KUKA KRL program: EPS_2_25252_SD6A_A_20250911081714.src

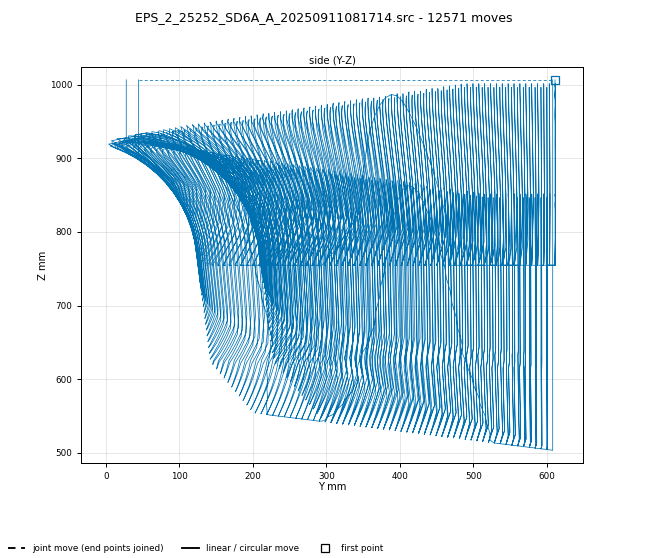
[picture p0: tool path of EPS_2_25252_SD6A_A_20250911081714.src, 12571 of 12573 moves have a stored position in this frame; points joined in program order, loops and branches not executed]
&ACCESS RVP
&REL 4
&COMMENT QRS 19112012
&PARAM EDITMASK = *
DEF PART()
EXT BAS (BAS_COMMAND :IN,REAL :IN )
INT I
BAS (#INITMOV,0 )

;KUKA QRS Post kuka4.cps  Date:22-06-2017 !

File_ID=2841

QRS_PRE_INIT()

;Init var - Until changes are made in qrs_pre_init
Outlet_Square_prg=0
Inlet_1_Square_prg=0
Inlet_2_Square_prg=0
Inlet_3_Square_prg=0
Inlet_4_Square_prg=0
Inlet_5_Square_prg=0

Outlet_1={X 0.000, Y 489.850, Z 814.000, B 0.000, E1 0.000 }
Inlet_1={X 0.000, Y 516.730, Z 721.500, B 0.000, E1 160.000 }
Outlet_1_type=366
Inlet_1_type=201
;QRS#1=Sidecore dimensions
;QRS#2=375-15" PVC SDR 35
;QRS#3=200-8" PVC SDR 35
;QRS#4=
;QRS#5=
;QRS#6=
;QRS#7=
;QRS#8=
;QRS#9=20Y PSX
;QRS#10=12-08 PSX
;QRS#11=
;QRS#12=
;QRS#13=
;QRS#14=
;QRS#15=
;QRS#16=1220x127x1295 4,25'
;QRS#17=EPS Height
;QRS#18=997
;QRS#19=*
;QRS#20= UPDATED VERSION 22-06-2017
;QRS#21=*
Outlet_Square=0250
Inlet_1_Square=0100
Inlet_2_Square=0
Inlet_3_Square=0
Inlet_4_Square=0
Inlet_5_Square=0
Mill_Square=1
Outlet_Square_Prg=252
Inlet_1_Square_prg=204

QRS_INIT()

$ADVANCE=5

; T1
PTP {E1 177.287,E2 177.287}
PTP {X 0,Y 611.066,A -85,B 0,C 180,E1 177.287,E2 177.287,E3 0,E4 0,E5 0,E6 0}
QRS_SPEED_INIT()
LIN {X 0,Y 611.066,Z 1007,A -85,B 0,C 180,E1 177.287,E2 177.287,E3 0,E4 0,E5 0,E6 0} C_VEL
LIN {X 0,Y 611.066,Z 756.81,A -85,B 0,C 180,E1 177.287,E2 177.287} C_VEL
LIN {X 0,Y 611.138,Z 754.81,A -85,B 0,C 180,E1 177.474,E2 177.474} C_VEL
LIN {X 0,Y 611.86,Z 754.81,A -85,B 0,C 180,E1 178.833,E2 178.833} C_VEL
LIN {X 0,Y 611.81,Z 754.81,A -85,B 0,C 180,E1 185.845,E2 185.845} C_VEL
LIN {X 0,Y 611.809,Z 754.81,A -85,B 0,C 180,E1 192.947,E2 192.947} C_VEL
LIN {X 0,Y 611.774,Z 754.81,A -85,B 0,C 180,E1 200.26,E2 200.26} C_VEL
LIN {X 0,Y 611.796,Z 754.81,A -85,B 0,C 180,E1 207.935,E2 207.935} C_VEL
LIN {X 0,Y 610.461,Z 754.81,A -85,B 0,C 180,E1 210.686,E2 210.686} C_VEL
LIN {X 0,Y 611.788,Z 754.81,A -85,B 0,C 180,E1 216.206,E2 216.206} C_VEL
LIN {X 0,Y 611.203,Z 754.81,A -85,B 0,C 180,E1 217.339,E2 217.339} C_VEL
LIN {X 0,Y 610.736,Z 754.81,A -85,B 0,C 180,E1 222.324,E2 222.324} C_VEL
LIN {X 0,Y 611.764,Z 754.81,A -85,B 0,C 180,E1 224.532,E2 224.532} C_VEL
LIN {X 0,Y 611.743,Z 754.81,A -85,B 0,C 180,E1 232.602,E2 232.602} C_VEL
LIN {X 0,Y 611.207,Z 754.81,A -85,B 0,C 180,E1 233.759,E2 233.759} C_VEL
LIN {X 0,Y 611.694,Z 754.81,A -85,B 0,C 180,E1 241.163,E2 241.163} C_VEL
LIN {X 0,Y 611.5,Z 754.81,A -85,B 0,C 180,E1 242.054,E2 242.054} C_VEL
LIN {X 0,Y 611.785,Z 754.81,A -85,B 0,C 180,E1 248.628,E2 248.628} C_VEL
LIN {X 0,Y 610.978,Z 754.81,A -85,B 0,C 180,E1 248.985,E2 248.985} C_VEL
LIN {X 0,Y 610.824,Z 754.81,A -85,B 0,C 180,E1 249.003,E2 249.003} C_VEL
LIN {X 0,Y 611.647,Z 795.005,A -85,B 0,C 180,E1 249.534,E2 249.534} C_VEL
LIN {X 0,Y 611.812,Z 820.275,A -85,B 0,C 180,E1 249.861,E2 249.861} C_VEL
LIN {X 0,Y 611.831,Z 829.389,A -85,B 0,C 180,E1 250.017,E2 250.017} C_VEL
LIN {X 0,Y 611.809,Z 838.409,A -85,B 0,C 180,E1 250.21,E2 250.21} C_VEL
LIN {X 0,Y 611.672,Z 847.342,A -85,B 0,C 180,E1 250.438,E2 250.438} C_VEL
LIN {X 0,Y 611.791,Z 856.186,A -85,B 0,C 180,E1 250.713,E2 250.713} C_VEL
LIN {X 0,Y 611.791,Z 863.938,A -85,B 0,C 180,E1 250.983,E2 250.983} C_VEL
LIN {X 0,Y 611.787,Z 873.56,A -85,B 0,C 180,E1 251.368,E2 251.368} C_VEL
LIN {X 0,Y 611.803,Z 882.055,A -85,B 0,C 180,E1 251.753,E2 251.753} C_VEL
LIN {X 0,Y 611.728,Z 891.103,A -85,B 0,C 180,E1 252.211,E2 252.211} C_VEL
LIN {X 0,Y 611.707,Z 900.538,A -85,B 0,C 180,E1 252.749,E2 252.749} C_VEL
LIN {X 0,Y 611.545,Z 908.953,A -85,B 0,C 180,E1 253.278,E2 253.278} C_VEL
LIN {X 0,Y 611.447,Z 915.387,A -85,B 0,C 180,E1 253.72,E2 253.72} C_VEL
LIN {X 0,Y 611.512,Z 922.82,A -85,B 0,C 180,E1 254.281,E2 254.281} C_VEL
LIN {X 0,Y 611.728,Z 930.719,A -85,B 0,C 180,E1 254.939,E2 254.939} C_VEL
LIN {X 0,Y 611.828,Z 937.206,A -85,B 0,C 180,E1 255.524,E2 255.524} C_VEL
LIN {X 0,Y 611.642,Z 944.107,A -85,B 0,C 180,E1 256.197,E2 256.197} C_VEL
LIN {X 0,Y 611.382,Z 950.111,A -85,B 0,C 180,E1 256.833,E2 256.833} C_VEL
LIN {X 0,Y 611.256,Z 955.826,A -85,B 0,C 180,E1 257.492,E2 257.492} C_VEL
LIN {X 0,Y 611.362,Z 961.718,A -85,B 0,C 180,E1 258.241,E2 258.241} C_VEL
LIN {X 0,Y 611.558,Z 966.083,A -85,B 0,C 180,E1 258.841,E2 258.841} C_VEL
LIN {X 0,Y 611.865,Z 971.956,A -85,B 0,C 180,E1 259.737,E2 259.737} C_VEL
LIN {X 0,Y 611.486,Z 977.196,A -85,B 0,C 180,E1 260.619,E2 260.619} C_VEL
LIN {X 0,Y 611.213,Z 980.408,A -85,B 0,C 180,E1 261.206,E2 261.206} C_VEL
LIN {X 0,Y 611.061,Z 984.692,A -85,B 0,C 180,E1 262.09,E2 262.09} C_VEL
LIN {X 0,Y 611.227,Z 988.443,A -85,B 0,C 180,E1 262.976,E2 262.976} C_VEL
LIN {X 0,Y 611.496,Z 990.636,A -85,B 0,C 180,E1 263.566,E2 263.566} C_VEL
LIN {X 0,Y 611.768,Z 992.621,A -85,B 0,C 180,E1 264.156,E2 264.156} C_VEL
LIN {X 0,Y 611.736,Z 994.457,A -85,B 0,C 180,E1 264.742,E2 264.742} C_VEL
LIN {X 0,Y 611.169,Z 997.433,A -85,B 0,C 180,E1 265.909,E2 265.909} C_VEL
LIN {X 0,Y 610.976,Z 998.684,A -85,B 0,C 180,E1 266.494,E2 266.494} C_VEL
LIN {X 0,Y 611.094,Z 1000.535,A -85,B 0,C 180,E1 267.713,E2 267.713} C_VEL
LIN {X 0,Y 611.599,Z 1001.553,A -85,B 0,C 180,E1 268.834,E2 268.834} C_VEL
LIN {X 0,Y 611.712,Z 1001.903,A -85,B 0,C 180,E1 269.768,E2 269.768} C_VEL
LIN {X 0,Y 611.468,Z 1001.915,A -85,B 0,C 180,E1 270.235,E2 270.235} C_VEL
LIN {X 0,Y 611.076,Z 1001.575,A -85,B 0,C 180,E1 271.17,E2 271.17} C_VEL
LIN {X 0,Y 611.004,Z 1000.586,A -85,B 0,C 180,E1 272.247,E2 272.247} C_VEL
LIN {X 0,Y 611.446,Z 998.665,A -85,B 0,C 180,E1 273.506,E2 273.506} C_VEL
LIN {X 0,Y 611.741,Z 997.407,A -85,B 0,C 180,E1 274.089,E2 274.089} C_VEL
LIN {X 0,Y 611.75,Z 996.021,A -85,B 0,C 180,E1 274.674,E2 274.674} C_VEL
LIN {X 0,Y 611.455,Z 994.46,A -85,B 0,C 180,E1 275.263,E2 275.263} C_VEL
LIN {X 0,Y 611.035,Z 991.688,A -85,B 0,C 180,E1 276.147,E2 276.147} C_VEL
LIN {X 0,Y 610.903,Z 988.434,A -85,B 0,C 180,E1 277.031,E2 277.031} C_VEL
LIN {X 0,Y 611.131,Z 984.681,A -85,B 0,C 180,E1 277.912,E2 277.912} C_VEL
LIN {X 0,Y 611.584,Z 980.396,A -85,B 0,C 180,E1 278.791,E2 278.791} C_VEL
LIN {X 0,Y 611.866,Z 977.182,A -85,B 0,C 180,E1 279.377,E2 279.377} C_VEL
LIN {X 0,Y 611.514,Z 971.941,A -85,B 0,C 180,E1 280.272,E2 280.272} C_VEL
LIN {X 0,Y 611.151,Z 964.994,A -85,B 0,C 180,E1 281.318,E2 281.318} C_VEL
LIN {X 0,Y 611.162,Z 959.425,A -85,B 0,C 180,E1 282.064,E2 282.064} C_VEL
LIN {X 0,Y 611.425,Z 953.292,A -85,B 0,C 180,E1 282.806,E2 282.806} C_VEL
LIN {X 0,Y 611.786,Z 945.803,A -85,B 0,C 180,E1 283.623,E2 283.623} C_VEL
LIN {X 0,Y 611.787,Z 939.857,A -85,B 0,C 180,E1 284.223,E2 284.223} C_VEL
LIN {X 0,Y 611.566,Z 932.74,A -85,B 0,C 180,E1 284.888,E2 284.888} C_VEL
LIN {X 0,Y 611.429,Z 926.124,A -85,B 0,C 180,E1 285.455,E2 285.455} C_VEL
LIN {X 0,Y 611.439,Z 919.137,A -85,B 0,C 180,E1 286.004,E2 286.004} C_VEL
LIN {X 0,Y 611.611,Z 911.498,A -85,B 0,C 180,E1 286.549,E2 286.549} C_VEL
LIN {X 0,Y 611.767,Z 903.322,A -85,B 0,C 180,E1 287.08,E2 287.08} C_VEL
LIN {X 0,Y 611.817,Z 895.304,A -85,B 0,C 180,E1 287.555,E2 287.555} C_VEL
LIN {X 0,Y 611.786,Z 886.651,A -85,B 0,C 180,E1 288.02,E2 288.02} C_VEL
LIN {X 0,Y 611.701,Z 878.735,A -85,B 0,C 180,E1 288.406,E2 288.406} C_VEL
LIN {X 0,Y 611.692,Z 869.834,A -85,B 0,C 180,E1 288.792,E2 288.792} C_VEL
LIN {X 0,Y 611.795,Z 859.549,A -85,B 0,C 180,E1 289.174,E2 289.174} C_VEL
LIN {X 0,Y 611.763,Z 849.942,A -85,B 0,C 180,E1 289.484,E2 289.484} C_VEL
LIN {X 0,Y 611.768,Z 843.149,A -85,B 0,C 180,E1 289.678,E2 289.678} C_VEL
LIN {X 0,Y 611.844,Z 831.276,A -85,B 0,C 180,E1 289.946,E2 289.946} C_VEL
LIN {X 0,Y 611.833,Z 821.432,A -85,B 0,C 180,E1 290.121,E2 290.121} C_VEL
LIN {X 0,Y 611.678,Z 798.302,A -85,B 0,C 180,E1 290.424,E2 290.424} C_VEL
LIN {X 0,Y 610.927,Z 760.221,A -85,B 0,C 180,E1 290.919,E2 290.919} C_VEL
LIN {X 0,Y 610.799,Z 754.81,A -85,B 0,C 180,E1 290.996,E2 290.996} C_VEL
LIN {X 0,Y 611.629,Z 754.81,A -85,B 0,C 180,E1 291.129,E2 291.129} C_VEL
LIN {X 0,Y 611.582,Z 754.81,A -85,B 0,C 180,E1 291.731,E2 291.731} C_VEL
LIN {X 0,Y 611.82,Z 754.81,A -85,B 0,C 180,E1 297.933,E2 297.933} C_VEL
LIN {X 0,Y 610.472,Z 754.81,A -85,B 0,C 180,E1 300.684,E2 300.684} C_VEL
LIN {X 0,Y 611.766,Z 754.81,A -85,B 0,C 180,E1 306.206,E2 306.206} C_VEL
LIN {X 0,Y 611.188,Z 754.81,A -85,B 0,C 180,E1 307.329,E2 307.329} C_VEL
LIN {X 0,Y 610.711,Z 754.81,A -85,B 0,C 180,E1 312.324,E2 312.324} C_VEL
LIN {X 0,Y 611.745,Z 754.81,A -85,B 0,C 180,E1 314.524,E2 314.524} C_VEL
LIN {X 0,Y 611.706,Z 754.81,A -85,B 0,C 180,E1 322.603,E2 322.603} C_VEL
LIN {X 0,Y 611.179,Z 754.81,A -85,B 0,C 180,E1 323.752,E2 323.752} C_VEL
LIN {X 0,Y 611.635,Z 754.81,A -85,B 0,C 180,E1 331.167,E2 331.167} C_VEL
LIN {X 0,Y 611.406,Z 754.81,A -85,B 0,C 180,E1 332.045,E2 332.045} C_VEL
LIN {X 0,Y 611.799,Z 754.81,A -85,B 0,C 180,E1 339.741,E2 339.741} C_VEL
LIN {X 0,Y 611.858,Z 754.81,A -85,B 0,C 180,E1 347.054,E2 347.054} C_VEL
LIN {X 0,Y 611.817,Z 754.81,A -85,B 0,C 180,E1 354.155,E2 354.155} C_VEL
LIN {X 0,Y 611.87,Z 754.81,A -85,B 0,C 180,E1 361.167,E2 361.167} C_VEL
LIN {X 0,Y 611.807,Z 754.81,A -85,B 0,C 180,E1 368.197,E2 368.197} C_VEL
LIN {X 0,Y 611.836,Z 754.81,A -85,B 0,C 180,E1 375.353,E2 375.353} C_VEL
LIN {X 0,Y 611.769,Z 754.81,A -85,B 0,C 180,E1 382.769,E2 382.769} C_VEL
LIN {X 0,Y 611.754,Z 754.81,A -85,B 0,C 180,E1 390.614,E2 390.614} C_VEL
LIN {X 0,Y 611.703,Z 754.81,A -85,B 0,C 180,E1 399.162,E2 399.162} C_VEL
LIN {X 0,Y 610.297,Z 754.81,A -85,B 0,C 180,E1 402.362,E2 402.362} C_VEL
LIN {X 0,Y 610.609,Z 754.81,A -85,B 0,C 180,E1 405.585,E2 405.585} C_VEL
LIN {X 0,Y 611.693,Z 754.81,A -85,B 0,C 180,E1 407.76,E2 407.76} C_VEL
LIN {X 0,Y 610.234,Z 754.81,A -85,B 0,C 180,E1 413.689,E2 413.689} C_VEL
LIN {X 0,Y 611.762,Z 754.81,A -85,B 0,C 180,E1 416.636,E2 416.636} C_VEL
LIN {X 0,Y 611.77,Z 754.81,A -85,B 0,C 180,E1 424.676,E2 424.676} C_VEL
LIN {X 0,Y 611.495,Z 754.81,A -85,B 0,C 180,E1 433.294,E2 433.294} C_VEL
LIN {X 0,Y 611.27,Z 754.81,A -85,B 0,C 180,E1 434.632,E2 434.632} C_VEL
LIN {X 0,Y 611.862,Z 754.81,A -85,B 0,C 180,E1 441.803,E2 441.803} C_VEL
LIN {X 0,Y 611.873,Z 754.81,A -85,B 0,C 180,E1 448.832,E2 448.832} C_VEL
LIN {X 0,Y 611.829,Z 754.81,A -85,B 0,C 180,E1 457.975,E2 457.975} C_VEL
LIN {X 0,Y 611.668,Z 754.904,A -85,B 0,C 180,E1 458.053,E2 458.053} C_VEL
LIN {X 0,Y 611.818,Z 763.461,A -85,B 0,C 180,E1 458.305,E2 458.305} C_VEL
LIN {X 0,Y 611.721,Z 770.819,A -85,B 0,C 180,E1 458.565,E2 458.565} C_VEL
LIN {X 0,Y 611.704,Z 779.374,A -85,B 0,C 180,E1 458.934,E2 458.934} C_VEL
LIN {X 0,Y 611.785,Z 786.58,A -85,B 0,C 180,E1 459.302,E2 459.302} C_VEL
LIN {X 0,Y 611.823,Z 794.066,A -85,B 0,C 180,E1 459.745,E2 459.745} C_VEL
LIN {X 0,Y 611.7,Z 801.675,A -85,B 0,C 180,E1 460.266,E2 460.266} C_VEL
LIN {X 0,Y 611.527,Z 809.163,A -85,B 0,C 180,E1 460.863,E2 460.863} C_VEL
LIN {X 0,Y 611.583,Z 813.985,A -85,B 0,C 180,E1 461.308,E2 461.308} C_VEL
LIN {X 0,Y 611.754,Z 819.881,A -85,B 0,C 180,E1 461.9,E2 461.9} C_VEL
LIN {X 0,Y 611.847,Z 825.006,A -85,B 0,C 180,E1 462.495,E2 462.495} C_VEL
LIN {X 0,Y 611.571,Z 830.05,A -85,B 0,C 180,E1 463.153,E2 463.153} C_VEL
LIN {X 0,Y 611.352,Z 834.118,A -85,B 0,C 180,E1 463.768,E2 463.768} C_VEL
LIN {X 0,Y 611.348,Z 837.585,A -85,B 0,C 180,E1 464.364,E2 464.364} C_VEL
LIN {X 0,Y 611.521,Z 840.61,A -85,B 0,C 180,E1 464.959,E2 464.959} C_VEL
LIN {X 0,Y 611.855,Z 843.98,A -85,B 0,C 180,E1 465.744,E2 465.744} C_VEL
LIN {X 0,Y 611.76,Z 845.466,A -85,B 0,C 180,E1 466.141,E2 466.141} C_VEL
LIN {X 0,Y 611.48,Z 847.279,A -85,B 0,C 180,E1 466.702,E2 466.702} C_VEL
LIN {X 0,Y 611.285,Z 848.511,A -85,B 0,C 180,E1 467.155,E2 467.155} C_VEL
LIN {X 0,Y 611.186,Z 849.953,A -85,B 0,C 180,E1 467.805,E2 467.805} C_VEL
LIN {X 0,Y 611.315,Z 850.927,A -85,B 0,C 180,E1 468.416,E2 468.416} C_VEL
LIN {X 0,Y 611.592,Z 851.56,A -85,B 0,C 180,E1 469.024,E2 469.024} C_VEL
LIN {X 0,Y 611.86,Z 851.874,A -85,B 0,C 180,E1 469.633,E2 469.633} C_VEL
LIN {X 0,Y 611.627,Z 851.891,A -85,B 0,C 180,E1 470.262,E2 470.262} C_VEL
LIN {X 0,Y 611.328,Z 851.62,A -85,B 0,C 180,E1 470.821,E2 470.821} C_VEL
LIN {X 0,Y 611.148,Z 851.071,A -85,B 0,C 180,E1 471.378,E2 471.378} C_VEL
LIN {X 0,Y 611.149,Z 849.995,A -85,B 0,C 180,E1 472.081,E2 472.081} C_VEL
LIN {X 0,Y 611.419,Z 848.438,A -85,B 0,C 180,E1 472.78,E2 472.78} C_VEL
LIN {X 0,Y 611.84,Z 846.085,A -85,B 0,C 180,E1 473.578,E2 473.578} C_VEL
LIN {X 0,Y 611.755,Z 844.446,A -85,B 0,C 180,E1 474.043,E2 474.043} C_VEL
LIN {X 0,Y 611.36,Z 840.812,A -85,B 0,C 180,E1 474.912,E2 474.912} C_VEL
LIN {X 0,Y 611.234,Z 837.514,A -85,B 0,C 180,E1 475.56,E2 475.56} C_VEL
LIN {X 0,Y 611.357,Z 833.768,A -85,B 0,C 180,E1 476.199,E2 476.199} C_VEL
LIN {X 0,Y 611.664,Z 829.491,A -85,B 0,C 180,E1 476.833,E2 476.833} C_VEL
LIN {X 0,Y 611.854,Z 826.255,A -85,B 0,C 180,E1 477.262,E2 477.262} C_VEL
LIN {X 0,Y 611.7,Z 820.546,A -85,B 0,C 180,E1 477.936,E2 477.936} C_VEL
LIN {X 0,Y 611.506,Z 814.309,A -85,B 0,C 180,E1 478.572,E2 478.572} C_VEL
LIN {X 0,Y 611.468,Z 809.884,A -85,B 0,C 180,E1 478.986,E2 478.986} C_VEL
LIN {X 0,Y 611.642,Z 803.331,A -85,B 0,C 180,E1 479.52,E2 479.52} C_VEL
LIN {X 0,Y 611.818,Z 795.711,A -85,B 0,C 180,E1 480.057,E2 480.057} C_VEL
LIN {X 0,Y 611.78,Z 788.564,A -85,B 0,C 180,E1 480.498,E2 480.498} C_VEL
LIN {X 0,Y 611.615,Z 780.628,A -85,B 0,C 180,E1 480.917,E2 480.917} C_VEL
LIN {X 0,Y 611.602,Z 773.495,A -85,B 0,C 180,E1 481.239,E2 481.239} C_VEL
LIN {X 0,Y 611.747,Z 764.95,A -85,B 0,C 180,E1 481.558,E2 481.558} C_VEL
LIN {X 0,Y 611.758,Z 755.735,A -85,B 0,C 180,E1 481.833,E2 481.833} C_VEL
LIN {X 0,Y 611.697,Z 754.81,A -85,B 0,C 180,E1 481.867,E2 481.867} C_VEL
LIN {X 0,Y 611.77,Z 754.81,A -85,B 0,C 180,E1 489.152,E2 489.152} C_VEL
LIN {X 0,Y 610.356,Z 754.81,A -85,B 0,C 180,E1 492.351,E2 492.351} C_VEL
LIN {X 0,Y 610.67,Z 754.81,A -85,B 0,C 180,E1 495.572,E2 495.572} C_VEL
LIN {X 0,Y 611.767,Z 754.81,A -85,B 0,C 180,E1 497.764,E2 497.764} C_VEL
LIN {X 0,Y 610.275,Z 754.81,A -85,B 0,C 180,E1 503.69,E2 503.69} C_VEL
LIN {X 0,Y 611.79,Z 754.81,A -85,B 0,C 180,E1 506.636,E2 506.636} C_VEL
LIN {X 0,Y 611.824,Z 754.81,A -85,B 0,C 180,E1 514.677,E2 514.677} C_VEL
LIN {X 0,Y 611.477,Z 754.81,A -85,B 0,C 180,E1 523.279,E2 523.279} C_VEL
LIN {X 0,Y 611.227,Z 754.81,A -85,B 0,C 180,E1 524.631,E2 524.631} C_VEL
LIN {X 0,Y 611.802,Z 754.81,A -85,B 0,C 180,E1 531.803,E2 531.803} C_VEL
LIN {X 0,Y 611.138,Z 754.81,A -85,B 0,C 180,E1 537.474,E2 537.474} C_VEL
LIN {X 0,Y 602.939,Z 754.81,A -85,B 0,C 180,E1 540.753,E2 540.753} C_VEL
LIN {X 0,Y 602.827,Z 754.81,A -85,B 0,C 180,E1 547.957,E2 547.957} C_VEL
LIN {X 0,Y 602.702,Z 754.81,A -85,B 0,C 180,E1 555.328,E2 555.328} C_VEL
LIN {X 0,Y 603.089,Z 754.81,A -85,B 0,C 180,E1 561.397,E2 561.397} C_VEL
LIN {X 0,Y 602.77,Z 754.81,A -85,B 0,C 180,E1 569.705,E2 569.705} C_VEL
LIN {X 0,Y 603.072,Z 754.81,A -85,B 0,C 180,E1 577.565,E2 577.565} C_VEL
LIN {X 0,Y 602.786,Z 754.81,A -85,B 0,C 180,E1 586.185,E2 586.185} C_VEL
LIN {X 0,Y 603.196,Z 754.81,A -85,B 0,C 180,E1 593.756,E2 593.756} C_VEL
LIN {X 0,Y 602.95,Z 754.81,A -85,B 0,C 180,E1 603.311,E2 603.311} C_VEL
LIN {X 0,Y 603.355,Z 756.25,A -85,B 0,C 180,E1 608.756,E2 608.756} C_VEL
LIN {X 0,Y 604.125,Z 848.863,A -85,B 0,C 180,E1 610.228,E2 610.228} C_VEL
LIN {X 0,Y 603.994,Z 900.949,A -85,B 0,C 180,E1 612.547,E2 612.547} C_VEL
LIN {X 0,Y 603.809,Z 944.075,A -85,B 0,C 180,E1 616.011,E2 616.011} C_VEL
LIN {X 0,Y 603.502,Z 977.731,A -85,B 0,C 180,E1 620.593,E2 620.593} C_VEL
LIN {X 0,Y 603.275,Z 997.05,A -85,B 0,C 180,E1 625.672,E2 625.672} C_VEL
LIN {X 0,Y 603.271,Z 1001.839,A -85,B 0,C 180,E1 630.721,E2 630.721} C_VEL
LIN {X 0,Y 603.203,Z 993.115,A -85,B 0,C 180,E1 635.776,E2 635.776} C_VEL
LIN {X 0,Y 603.407,Z 970.196,A -85,B 0,C 180,E1 640.69,E2 640.69} C_VEL
LIN {X 0,Y 603.74,Z 934.098,A -85,B 0,C 180,E1 644.965,E2 644.965} C_VEL
LIN {X 0,Y 604.102,Z 887.651,A -85,B 0,C 180,E1 648.207,E2 648.207} C_VEL
LIN {X 0,Y 604.321,Z 835.988,A -85,B 0,C 180,E1 650.104,E2 650.104} C_VEL
LIN {X 0,Y 603.622,Z 754.81,A -85,B 0,C 180,E1 651.38,E2 651.38} C_VEL
LIN {X 0,Y 602.793,Z 754.81,A -85,B 0,C 180,E1 659.713,E2 659.713} C_VEL
LIN {X 0,Y 603.053,Z 754.81,A -85,B 0,C 180,E1 667.566,E2 667.566} C_VEL
LIN {X 0,Y 602.757,Z 754.81,A -85,B 0,C 180,E1 676.185,E2 676.185} C_VEL
LIN {X 0,Y 603.175,Z 754.81,A -85,B 0,C 180,E1 683.757,E2 683.757} C_VEL
LIN {X 0,Y 603.254,Z 754.81,A -85,B 0,C 180,E1 692.267,E2 692.267} C_VEL
LIN {X 0,Y 602.853,Z 754.81,A -85,B 0,C 180,E1 701.662,E2 701.662} C_VEL
LIN {X 0,Y 602.898,Z 754.81,A -85,B 0,C 180,E1 709.12,E2 709.12} C_VEL
LIN {X 0,Y 602.842,Z 754.81,A -85,B 0,C 180,E1 716.394,E2 716.394} C_VEL
LIN {X 0,Y 602.808,Z 754.81,A -85,B 0,C 180,E1 723.61,E2 723.61} C_VEL
LIN {X 0,Y 603.164,Z 754.81,A -85,B 0,C 180,E1 729.414,E2 729.414} C_VEL
LIN {X 0,Y 603.021,Z 754.81,A -85,B 0,C 180,E1 736.824,E2 736.824} C_VEL
LIN {X 0,Y 602.77,Z 754.81,A -85,B 0,C 180,E1 744.547,E2 744.547} C_VEL
LIN {X 0,Y 602.582,Z 754.81,A -85,B 0,C 180,E1 752.468,E2 752.468} C_VEL
LIN {X 0,Y 603.22,Z 754.81,A -85,B 0,C 180,E1 759.907,E2 759.907} C_VEL
LIN {X 0,Y 603.356,Z 754.81,A -85,B 0,C 180,E1 768.199,E2 768.199} C_VEL
LIN {X 0,Y 603.218,Z 754.81,A -85,B 0,C 180,E1 777.438,E2 777.438} C_VEL
LIN {X 0,Y 603.153,Z 754.81,A -85,B 0,C 180,E1 785.471,E2 785.471} C_VEL
LIN {X 0,Y 603.238,Z 754.81,A -85,B 0,C 180,E1 794.683,E2 794.683} C_VEL
LIN {X 0,Y 602.911,Z 754.81,A -85,B 0,C 180,E1 803.858,E2 803.858} C_VEL
LIN {X 0,Y 602.597,Z 754.81,A -85,B 0,C 180,E1 810.721,E2 810.721} C_VEL
LIN {X 0,Y 603.88,Z 756.612,A -85,B 0,C 180,E1 817.944,E2 817.944} C_VEL
LIN {X 0,Y 603.91,Z 796.409,A -85,B 0,C 180,E1 819.765,E2 819.765} C_VEL
LIN {X 0,Y 603.782,Z 827.416,A -85,B 0,C 180,E1 822.704,E2 822.704} C_VEL
LIN {X 0,Y 603.602,Z 846.583,A -85,B 0,C 180,E1 826.43,E2 826.43} C_VEL
LIN {X 0,Y 603.782,Z 851.979,A -85,B 0,C 180,E1 829.835,E2 829.835} C_VEL
LIN {X 0,Y 603.782,Z 845.084,A -85,B 0,C 180,E1 833.93,E2 833.93} C_VEL
LIN {X 0,Y 603.788,Z 823.442,A -85,B 0,C 180,E1 837.709,E2 837.709} C_VEL
LIN {X 0,Y 603.91,Z 790.475,A -85,B 0,C 180,E1 840.522,E2 840.522} C_VEL
LIN {X 0,Y 603.494,Z 754.81,A -85,B 0,C 180,E1 842.194,E2 842.194} C_VEL
LIN {X 0,Y 603.287,Z 754.81,A -85,B 0,C 180,E1 849.9,E2 849.9} C_VEL
LIN {X 0,Y 603.418,Z 754.81,A -85,B 0,C 180,E1 858.204,E2 858.204} C_VEL
LIN {X 0,Y 603.274,Z 754.81,A -85,B 0,C 180,E1 867.427,E2 867.427} C_VEL
LIN {X 0,Y 603.227,Z 754.81,A -85,B 0,C 180,E1 875.473,E2 875.473} C_VEL
LIN {X 0,Y 603.194,Z 754.81,A -85,B 0,C 180,E1 884.681,E2 884.681} C_VEL
LIN {X 0,Y 602.878,Z 754.81,A -85,B 0,C 180,E1 893.875,E2 893.875} C_VEL
LIN {X 0,Y 602.939,Z 754.81,A -85,B 0,C 180,E1 900.753,E2 900.753} C_VEL
LIN {X 0,Y 594.952,Z 754.81,A -85,B 0,C 180,E1 904.052,E2 904.052} C_VEL
LIN {X 0,Y 595.421,Z 754.81,A -85,B 0,C 180,E1 912.51,E2 912.51} C_VEL
LIN {X 0,Y 594.956,Z 754.81,A -85,B 0,C 180,E1 921.704,E2 921.704} C_VEL
LIN {X 0,Y 594.736,Z 754.81,A -85,B 0,C 180,E1 929.837,E2 929.837} C_VEL
LIN {X 0,Y 595.425,Z 754.81,A -85,B 0,C 180,E1 936.792,E2 936.792} C_VEL
LIN {X 0,Y 595.044,Z 754.81,A -85,B 0,C 180,E1 945.465,E2 945.465} C_VEL
LIN {X 0,Y 595.255,Z 754.81,A -85,B 0,C 180,E1 953.421,E2 953.421} C_VEL
LIN {X 0,Y 595.313,Z 754.81,A -85,B 0,C 180,E1 961.862,E2 961.862} C_VEL
LIN {X 0,Y 595.708,Z 756.326,A -85,B 0,C 180,E1 968.471,E2 968.471} C_VEL
LIN {X 0,Y 596.585,Z 848.864,A -85,B 0,C 180,E1 969.967,E2 969.967} C_VEL
LIN {X 0,Y 596.304,Z 900.979,A -85,B 0,C 180,E1 972.316,E2 972.316} C_VEL
LIN {X 0,Y 595.976,Z 944.04,A -85,B 0,C 180,E1 975.82,E2 975.82} C_VEL
LIN {X 0,Y 595.729,Z 975.748,A -85,B 0,C 180,E1 980.099,E2 980.099} C_VEL
LIN {X 0,Y 595.635,Z 995.224,A -85,B 0,C 180,E1 984.884,E2 984.884} C_VEL
LIN {X 0,Y 595.643,Z 1001.839,A -85,B 0,C 180,E1 989.271,E2 989.271} C_VEL
LIN {X 0,Y 595.742,Z 997.049,A -85,B 0,C 180,E1 994.383,E2 994.383} C_VEL
LIN {X 0,Y 595.9,Z 977.727,A -85,B 0,C 180,E1 999.529,E2 999.529} C_VEL
LIN {X 0,Y 596.013,Z 945.729,A -85,B 0,C 180,E1 1003.999,E2 1003.999} C_VEL
LIN {X 0,Y 596.367,Z 901.589,A -85,B 0,C 180,E1 1007.644,E2 1007.644} C_VEL
LIN {X 0,Y 596.659,Z 850.037,A -85,B 0,C 180,E1 1009.995,E2 1009.995} C_VEL
LIN {X 0,Y 595.986,Z 759.919,A -85,B 0,C 180,E1 1011.473,E2 1011.473} C_VEL
LIN {X 0,Y 595.487,Z 754.81,A -85,B 0,C 180,E1 1011.687,E2 1011.687} C_VEL
LIN {X 0,Y 594.758,Z 754.81,A -85,B 0,C 180,E1 1019.839,E2 1019.839} C_VEL
LIN {X 0,Y 595.42,Z 754.81,A -85,B 0,C 180,E1 1026.796,E2 1026.796} C_VEL
LIN {X 0,Y 595.018,Z 754.81,A -85,B 0,C 180,E1 1035.466,E2 1035.466} C_VEL
LIN {X 0,Y 595.232,Z 754.81,A -85,B 0,C 180,E1 1043.429,E2 1043.429} C_VEL
LIN {X 0,Y 595.205,Z 754.81,A -85,B 0,C 180,E1 1051.859,E2 1051.859} C_VEL
LIN {X 0,Y 594.941,Z 754.81,A -85,B 0,C 180,E1 1061.409,E2 1061.409} C_VEL
LIN {X 0,Y 594.918,Z 754.81,A -85,B 0,C 180,E1 1069.144,E2 1069.144} C_VEL
LIN {X 0,Y 594.853,Z 754.81,A -85,B 0,C 180,E1 1076.345,E2 1076.345} C_VEL
LIN {X 0,Y 594.797,Z 754.81,A -85,B 0,C 180,E1 1083.659,E2 1083.659} C_VEL
LIN {X 0,Y 594.754,Z 754.81,A -85,B 0,C 180,E1 1090.773,E2 1090.773} C_VEL
LIN {X 0,Y 594.921,Z 754.81,A -85,B 0,C 180,E1 1097.06,E2 1097.06} C_VEL
LIN {X 0,Y 594.608,Z 754.81,A -85,B 0,C 180,E1 1105.035,E2 1105.035} C_VEL
LIN {X 0,Y 595.098,Z 754.81,A -85,B 0,C 180,E1 1111.52,E2 1111.52} C_VEL
LIN {X 0,Y 594.624,Z 754.81,A -85,B 0,C 180,E1 1121.158,E2 1121.158} C_VEL
LIN {X 0,Y 594.642,Z 754.81,A -85,B 0,C 180,E1 1129.399,E2 1129.399} C_VEL
LIN {X 0,Y 594.722,Z 754.81,A -85,B 0,C 180,E1 1138.459,E2 1138.459} C_VEL
LIN {X 0,Y 594.469,Z 754.81,A -85,B 0,C 180,E1 1146.691,E2 1146.691} C_VEL
LIN {X 0,Y 595.236,Z 754.81,A -85,B 0,C 180,E1 1154.472,E2 1154.472} C_VEL
LIN {X 0,Y 595.047,Z 754.81,A -85,B 0,C 180,E1 1163.409,E2 1163.409} C_VEL
LIN {X 0,Y 594.586,Z 754.81,A -85,B 0,C 180,E1 1170.731,E2 1170.731} C_VEL
LIN {X 0,Y 595.813,Z 756.512,A -85,B 0,C 180,E1 1177.776,E2 1177.776} C_VEL
LIN {X 0,Y 596.015,Z 796.255,A -85,B 0,C 180,E1 1179.618,E2 1179.618} C_VEL
LIN {X 0,Y 595.814,Z 828.021,A -85,B 0,C 180,E1 1182.69,E2 1182.69} C_VEL
LIN {X 0,Y 595.5,Z 847.425,A -85,B 0,C 180,E1 1186.66,E2 1186.66} C_VEL
LIN {X 0,Y 595.63,Z 851.97,A -85,B 0,C 180,E1 1190.118,E2 1190.118} C_VEL
LIN {X 0,Y 595.655,Z 843.869,A -85,B 0,C 180,E1 1194.318,E2 1194.318} C_VEL
LIN {X 0,Y 595.748,Z 820.861,A -85,B 0,C 180,E1 1198.115,E2 1198.115} C_VEL
LIN {X 0,Y 595.954,Z 786.961,A -85,B 0,C 180,E1 1200.873,E2 1200.873} C_VEL
LIN {X 0,Y 595.408,Z 754.81,A -85,B 0,C 180,E1 1202.342,E2 1202.342} C_VEL
LIN {X 0,Y 594.679,Z 754.81,A -85,B 0,C 180,E1 1211.163,E2 1211.163} C_VEL
LIN {X 0,Y 594.689,Z 754.81,A -85,B 0,C 180,E1 1219.402,E2 1219.402} C_VEL
LIN {X 0,Y 594.782,Z 754.81,A -85,B 0,C 180,E1 1228.461,E2 1228.461} C_VEL
LIN {X 0,Y 594.507,Z 754.81,A -85,B 0,C 180,E1 1236.691,E2 1236.691} C_VEL
LIN {X 0,Y 595.199,Z 754.81,A -85,B 0,C 180,E1 1244.47,E2 1244.47} C_VEL
LIN {X 0,Y 595.012,Z 754.81,A -85,B 0,C 180,E1 1253.408,E2 1253.408} C_VEL
LIN {X 0,Y 594.958,Z 754.81,A -85,B 0,C 180,E1 1260.731,E2 1260.731} C_VEL
LIN {X 0,Y 594.952,Z 754.81,A -85,B 0,C 180,E1 1264.052,E2 1264.052} C_VEL
LIN {X 0,Y 587.035,Z 754.81,A -85,B 0,C 180,E1 1267.425,E2 1267.425} C_VEL
LIN {X 0,Y 587.105,Z 754.81,A -85,B 0,C 180,E1 1274.232,E2 1274.232} C_VEL
LIN {X 0,Y 586.825,Z 754.81,A -85,B 0,C 180,E1 1282.021,E2 1282.021} C_VEL
LIN {X 0,Y 586.579,Z 754.81,A -85,B 0,C 180,E1 1290.295,E2 1290.295} C_VEL
LIN {X 0,Y 586.872,Z 754.81,A -85,B 0,C 180,E1 1297.937,E2 1297.937} C_VEL
LIN {X 0,Y 586.578,Z 754.81,A -85,B 0,C 180,E1 1306.718,E2 1306.718} C_VEL
LIN {X 0,Y 586.764,Z 754.81,A -85,B 0,C 180,E1 1314.553,E2 1314.553} C_VEL
LIN {X 0,Y 586.949,Z 754.81,A -85,B 0,C 180,E1 1323.12,E2 1323.12} C_VEL
LIN {X 0,Y 587.567,Z 756.444,A -85,B 0,C 180,E1 1328.159,E2 1328.159} C_VEL
LIN {X 0,Y 589.058,Z 849.901,A -85,B 0,C 180,E1 1329.731,E2 1329.731} C_VEL
LIN {X 0,Y 588.579,Z 901.19,A -85,B 0,C 180,E1 1332.089,E2 1332.089} C_VEL
LIN {X 0,Y 588.134,Z 944.29,A -85,B 0,C 180,E1 1335.654,E2 1335.654} C_VEL
LIN {X 0,Y 587.65,Z 977.732,A -85,B 0,C 180,E1 1340.337,E2 1340.337} C_VEL
LIN {X 0,Y 587.32,Z 997.051,A -85,B 0,C 180,E1 1345.555,E2 1345.555} C_VEL
LIN {X 0,Y 587.26,Z 1001.839,A -85,B 0,C 180,E1 1350.741,E2 1350.741} C_VEL
LIN {X 0,Y 587.241,Z 993.533,A -85,B 0,C 180,E1 1355.798,E2 1355.798} C_VEL
LIN {X 0,Y 587.505,Z 971.486,A -85,B 0,C 180,E1 1360.775,E2 1360.775} C_VEL
LIN {X 0,Y 588.046,Z 935.848,A -85,B 0,C 180,E1 1365.21,E2 1365.21} C_VEL
LIN {X 0,Y 588.767,Z 889.465,A -85,B 0,C 180,E1 1368.601,E2 1368.601} C_VEL
LIN {X 0,Y 589.291,Z 837.458,A -85,B 0,C 180,E1 1370.603,E2 1370.603} C_VEL
LIN {X 0,Y 587.351,Z 754.81,A -85,B 0,C 180,E1 1372.003,E2 1372.003} C_VEL
LIN {X 0,Y 586.622,Z 754.81,A -85,B 0,C 180,E1 1380.296,E2 1380.296} C_VEL
LIN {X 0,Y 586.86,Z 754.81,A -85,B 0,C 180,E1 1387.94,E2 1387.94} C_VEL
LIN {X 0,Y 586.55,Z 754.81,A -85,B 0,C 180,E1 1396.718,E2 1396.718} C_VEL
LIN {X 0,Y 586.717,Z 754.81,A -85,B 0,C 180,E1 1404.565,E2 1404.565} C_VEL
LIN {X 0,Y 586.719,Z 754.81,A -85,B 0,C 180,E1 1413.172,E2 1413.172} C_VEL
LIN {X 0,Y 586.99,Z 754.81,A -85,B 0,C 180,E1 1421.148,E2 1421.148} C_VEL
LIN {X 0,Y 586.996,Z 754.81,A -85,B 0,C 180,E1 1428.822,E2 1428.822} C_VEL
LIN {X 0,Y 586.863,Z 754.81,A -85,B 0,C 180,E1 1436.295,E2 1436.295} C_VEL
LIN {X 0,Y 586.788,Z 754.81,A -85,B 0,C 180,E1 1443.709,E2 1443.709} C_VEL
LIN {X 0,Y 587.08,Z 754.81,A -85,B 0,C 180,E1 1449.675,E2 1449.675} C_VEL
LIN {X 0,Y 586.837,Z 754.81,A -85,B 0,C 180,E1 1457.303,E2 1457.303} C_VEL
LIN {X 0,Y 586.552,Z 754.81,A -85,B 0,C 180,E1 1465.273,E2 1465.273} C_VEL
LIN {X 0,Y 586.481,Z 754.81,A -85,B 0,C 180,E1 1472.757,E2 1472.757} C_VEL
LIN {X 0,Y 586.582,Z 754.81,A -85,B 0,C 180,E1 1481.28,E2 1481.28} C_VEL
LIN {X 0,Y 586.979,Z 754.81,A -85,B 0,C 180,E1 1488.755,E2 1488.755} C_VEL
LIN {X 0,Y 586.793,Z 754.81,A -85,B 0,C 180,E1 1497.982,E2 1497.982} C_VEL
LIN {X 0,Y 586.445,Z 754.81,A -85,B 0,C 180,E1 1506.732,E2 1506.732} C_VEL
LIN {X 0,Y 587.211,Z 754.81,A -85,B 0,C 180,E1 1514.254,E2 1514.254} C_VEL
LIN {X 0,Y 587.076,Z 754.81,A -85,B 0,C 180,E1 1523.32,E2 1523.32} C_VEL
LIN {X 0,Y 586.573,Z 754.81,A -85,B 0,C 180,E1 1530.741,E2 1530.741} C_VEL
LIN {X 0,Y 587.516,Z 755.536,A -85,B 0,C 180,E1 1537.573,E2 1537.573} C_VEL
LIN {X 0,Y 588.143,Z 796.092,A -85,B 0,C 180,E1 1539.467,E2 1539.467} C_VEL
LIN {X 0,Y 587.93,Z 827.248,A -85,B 0,C 180,E1 1542.484,E2 1542.484} C_VEL
LIN {X 0,Y 587.586,Z 847.03,A -85,B 0,C 180,E1 1546.478,E2 1546.478} C_VEL
LIN {X 0,Y 587.515,Z 851.904,A -85,B 0,C 180,E1 1550.408,E2 1550.408} C_VEL
LIN {X 0,Y 587.62,Z 843.766,A -85,B 0,C 180,E1 1554.406,E2 1554.406} C_VEL
LIN {X 0,Y 587.791,Z 821.637,A -85,B 0,C 180,E1 1558.137,E2 1558.137} C_VEL
LIN {X 0,Y 588.062,Z 787.082,A -85,B 0,C 180,E1 1561.015,E2 1561.015} C_VEL
LIN {X 0,Y 587.36,Z 754.81,A -85,B 0,C 180,E1 1562.41,E2 1562.41} C_VEL
LIN {X 0,Y 586.64,Z 754.81,A -85,B 0,C 180,E1 1571.273,E2 1571.273} C_VEL
LIN {X 0,Y 587.064,Z 754.81,A -85,B 0,C 180,E1 1578.761,E2 1578.761} C_VEL
LIN {X 0,Y 586.843,Z 754.81,A -85,B 0,C 180,E1 1587.984,E2 1587.984} C_VEL
LIN {X 0,Y 586.489,Z 754.81,A -85,B 0,C 180,E1 1596.719,E2 1596.719} C_VEL
LIN {X 0,Y 587.177,Z 754.81,A -85,B 0,C 180,E1 1604.252,E2 1604.252} C_VEL
LIN {X 0,Y 587.045,Z 754.81,A -85,B 0,C 180,E1 1613.318,E2 1613.318} C_VEL
LIN {X 0,Y 586.953,Z 754.81,A -85,B 0,C 180,E1 1620.739,E2 1620.739} C_VEL
LIN {X 0,Y 587.035,Z 754.81,A -85,B 0,C 180,E1 1627.425,E2 1627.425} C_VEL
LIN {X 0,Y 578.821,Z 754.81,A -85,B 0,C 180,E1 1630.811,E2 1630.811} C_VEL
LIN {X 0,Y 579.054,Z 754.81,A -85,B 0,C 180,E1 1639.121,E2 1639.121} C_VEL
LIN {X 0,Y 579.026,Z 754.81,A -85,B 0,C 180,E1 1649.001,E2 1649.001} C_VEL
LIN {X 0,Y 578.852,Z 754.81,A -85,B 0,C 180,E1 1658.029,E2 1658.029} C_VEL
LIN {X 0,Y 578.746,Z 754.81,A -85,B 0,C 180,E1 1666.141,E2 1666.141} C_VEL
LIN {X 0,Y 578.844,Z 754.81,A -85,B 0,C 180,E1 1673.851,E2 1673.851} C_VEL
LIN {X 0,Y 578.988,Z 754.81,A -85,B 0,C 180,E1 1682.698,E2 1682.698} C_VEL
LIN {X 0,Y 579.35,Z 755.953,A -85,B 0,C 180,E1 1687.826,E2 1687.826} C_VEL
LIN {X 0,Y 581.581,Z 848.986,A -85,B 0,C 180,E1 1689.431,E2 1689.431} C_VEL
LIN {X 0,Y 580.89,Z 900.956,A -85,B 0,C 180,E1 1691.829,E2 1691.829} C_VEL
LIN {X 0,Y 580.283,Z 944.638,A -85,B 0,C 180,E1 1695.494,E2 1695.494} C_VEL
LIN {X 0,Y 579.711,Z 977.733,A -85,B 0,C 180,E1 1700.203,E2 1700.203} C_VEL
LIN {X 0,Y 579.367,Z 997.05,A -85,B 0,C 180,E1 1705.493,E2 1705.493} C_VEL
LIN {X 0,Y 579.265,Z 1001.838,A -85,B 0,C 180,E1 1710.751,E2 1710.751} C_VEL
LIN {X 0,Y 579.204,Z 993.534,A -85,B 0,C 180,E1 1715.879,E2 1715.879} C_VEL
LIN {X 0,Y 579.477,Z 970.786,A -85,B 0,C 180,E1 1721.043,E2 1721.043} C_VEL
LIN {X 0,Y 580.199,Z 934.751,A -85,B 0,C 180,E1 1725.527,E2 1725.527} C_VEL
LIN {X 0,Y 581.132,Z 887.661,A -85,B 0,C 180,E1 1728.954,E2 1728.954} C_VEL
LIN {X 0,Y 581.823,Z 834.061,A -85,B 0,C 180,E1 1730.965,E2 1730.965} C_VEL
LIN {X 0,Y 579.281,Z 754.81,A -85,B 0,C 180,E1 1732.231,E2 1732.231} C_VEL
LIN {X 0,Y 578.477,Z 754.81,A -85,B 0,C 180,E1 1740.769,E2 1740.769} C_VEL
LIN {X 0,Y 578.838,Z 754.81,A -85,B 0,C 180,E1 1748.033,E2 1748.033} C_VEL
LIN {X 0,Y 578.727,Z 754.81,A -85,B 0,C 180,E1 1756.148,E2 1756.148} C_VEL
LIN {X 0,Y 578.807,Z 754.81,A -85,B 0,C 180,E1 1763.851,E2 1763.851} C_VEL
LIN {X 0,Y 578.793,Z 754.81,A -85,B 0,C 180,E1 1772.69,E2 1772.69} C_VEL
LIN {X 0,Y 579.08,Z 754.81,A -85,B 0,C 180,E1 1780.88,E2 1780.88} C_VEL
LIN {X 0,Y 578.81,Z 754.81,A -85,B 0,C 180,E1 1789.488,E2 1789.488} C_VEL
LIN {X 0,Y 578.9,Z 754.81,A -85,B 0,C 180,E1 1796.244,E2 1796.244} C_VEL
LIN {X 0,Y 578.809,Z 754.81,A -85,B 0,C 180,E1 1803.76,E2 1803.76} C_VEL
LIN {X 0,Y 578.683,Z 754.81,A -85,B 0,C 180,E1 1811.345,E2 1811.345} C_VEL
LIN {X 0,Y 578.789,Z 754.81,A -85,B 0,C 180,E1 1817.551,E2 1817.551} C_VEL
LIN {X 0,Y 578.478,Z 754.81,A -85,B 0,C 180,E1 1825.651,E2 1825.651} C_VEL
LIN {X 0,Y 578.574,Z 754.81,A -85,B 0,C 180,E1 1832.529,E2 1832.529} C_VEL
LIN {X 0,Y 578.49,Z 754.81,A -85,B 0,C 180,E1 1841.612,E2 1841.612} C_VEL
LIN {X 0,Y 578.393,Z 754.81,A -85,B 0,C 180,E1 1849.997,E2 1849.997} C_VEL
LIN {X 0,Y 578.617,Z 754.81,A -85,B 0,C 180,E1 1858.475,E2 1858.475} C_VEL
LIN {X 0,Y 578.673,Z 754.81,A -85,B 0,C 180,E1 1866.015,E2 1866.015} C_VEL
LIN {X 0,Y 578.765,Z 754.81,A -85,B 0,C 180,E1 1875.575,E2 1875.575} C_VEL
LIN {X 0,Y 579.096,Z 754.81,A -85,B 0,C 180,E1 1883.227,E2 1883.227} C_VEL
LIN {X 0,Y 578.56,Z 754.81,A -85,B 0,C 180,E1 1890.751,E2 1890.751} C_VEL
LIN {X 0,Y 579.544,Z 756.488,A -85,B 0,C 180,E1 1897.428,E2 1897.428} C_VEL
LIN {X 0,Y 580.227,Z 797.325,A -85,B 0,C 180,E1 1899.408,E2 1899.408} C_VEL
LIN {X 0,Y 579.833,Z 829.239,A -85,B 0,C 180,E1 1902.661,E2 1902.661} C_VEL
LIN {X 0,Y 579.579,Z 847.25,A -85,B 0,C 180,E1 1906.504,E2 1906.504} C_VEL
LIN {X 0,Y 579.427,Z 851.758,A -85,B 0,C 180,E1 1910.706,E2 1910.706} C_VEL
LIN {X 0,Y 579.405,Z 841.642,A -85,B 0,C 180,E1 1914.998,E2 1914.998} C_VEL
LIN {X 0,Y 579.774,Z 817.414,A -85,B 0,C 180,E1 1918.731,E2 1918.731} C_VEL
LIN {X 0,Y 580.152,Z 782.28,A -85,B 0,C 180,E1 1921.436,E2 1921.436} C_VEL
LIN {X 0,Y 579.231,Z 754.81,A -85,B 0,C 180,E1 1922.69,E2 1922.69} C_VEL
LIN {X 0,Y 578.54,Z 754.81,A -85,B 0,C 180,E1 1931.616,E2 1931.616} C_VEL
LIN {X 0,Y 578.434,Z 754.81,A -85,B 0,C 180,E1 1939.999,E2 1939.999} C_VEL
LIN {X 0,Y 578.669,Z 754.81,A -85,B 0,C 180,E1 1948.464,E2 1948.464} C_VEL
LIN {X 0,Y 578.715,Z 754.81,A -85,B 0,C 180,E1 1956.016,E2 1956.016} C_VEL
LIN {X 0,Y 578.734,Z 754.81,A -85,B 0,C 180,E1 1965.573,E2 1965.573} C_VEL
LIN {X 0,Y 579.064,Z 754.81,A -85,B 0,C 180,E1 1973.225,E2 1973.225} C_VEL
LIN {X 0,Y 578.974,Z 754.81,A -85,B 0,C 180,E1 1980.749,E2 1980.749} C_VEL
LIN {X 0,Y 578.766,Z 754.81,A -85,B 0,C 180,E1 1988.29,E2 1988.29} C_VEL
LIN {X 0,Y 578.821,Z 754.81,A -85,B 0,C 180,E1 1990.811,E2 1990.811} C_VEL
LIN {X 0,Y 571.03,Z 754.81,A -85,B 0,C 180,E1 1994.284,E2 1994.284} C_VEL
LIN {X 0,Y 570.642,Z 754.81,A -85,B 0,C 180,E1 2002.679,E2 2002.679} C_VEL
LIN {X 0,Y 570.599,Z 754.81,A -85,B 0,C 180,E1 2010.189,E2 2010.189} C_VEL
LIN {X 0,Y 570.64,Z 754.81,A -85,B 0,C 180,E1 2018.676,E2 2018.676} C_VEL
LIN {X 0,Y 570.428,Z 754.81,A -85,B 0,C 180,E1 2027.281,E2 2027.281} C_VEL
LIN {X 0,Y 570.47,Z 754.81,A -85,B 0,C 180,E1 2035.114,E2 2035.114} C_VEL
LIN {X 0,Y 570.724,Z 754.81,A -85,B 0,C 180,E1 2043.977,E2 2043.977} C_VEL
LIN {X 0,Y 571.31,Z 756.347,A -85,B 0,C 180,E1 2047.502,E2 2047.502} C_VEL
LIN {X 0,Y 574.215,Z 789.478,A -85,B 0,C 180,E1 2048.061,E2 2048.061} C_VEL
LIN {X 0,Y 574.016,Z 854.655,A -85,B 0,C 180,E1 2049.332,E2 2049.332} C_VEL
LIN {X 0,Y 573.141,Z 905.505,A -85,B 0,C 180,E1 2051.874,E2 2051.874} C_VEL
LIN {X 0,Y 572.291,Z 948.096,A -85,B 0,C 180,E1 2055.673,E2 2055.673} C_VEL
LIN {X 0,Y 571.624,Z 979.692,A -85,B 0,C 180,E1 2060.449,E2 2060.449} C_VEL
LIN {X 0,Y 571.387,Z 997.05,A -85,B 0,C 180,E1 2065.43,E2 2065.43} C_VEL
LIN {X 0,Y 571.26,Z 1001.838,A -85,B 0,C 180,E1 2070.762,E2 2070.762} C_VEL
LIN {X 0,Y 571.137,Z 993.116,A -85,B 0,C 180,E1 2076.102,E2 2076.102} C_VEL
LIN {X 0,Y 571.528,Z 970.322,A -85,B 0,C 180,E1 2081.273,E2 2081.273} C_VEL
LIN {X 0,Y 572.328,Z 933.749,A -85,B 0,C 180,E1 2085.84,E2 2085.84} C_VEL
LIN {X 0,Y 573.477,Z 887.664,A -85,B 0,C 180,E1 2089.216,E2 2089.216} C_VEL
LIN {X 0,Y 574.362,Z 834.061,A -85,B 0,C 180,E1 2091.251,E2 2091.251} C_VEL
LIN {X 0,Y 571.765,Z 757.707,A -85,B 0,C 180,E1 2092.461,E2 2092.461} C_VEL
LIN {X 0,Y 571.145,Z 754.81,A -85,B 0,C 180,E1 2092.661,E2 2092.661} C_VEL
LIN {X 0,Y 570.626,Z 754.81,A -85,B 0,C 180,E1 2100.199,E2 2100.199} C_VEL
LIN {X 0,Y 570.617,Z 754.81,A -85,B 0,C 180,E1 2108.682,E2 2108.682} C_VEL
LIN {X 0,Y 570.378,Z 754.81,A -85,B 0,C 180,E1 2117.28,E2 2117.28} C_VEL
LIN {X 0,Y 570.437,Z 754.81,A -85,B 0,C 180,E1 2125.115,E2 2125.115} C_VEL
LIN {X 0,Y 570.718,Z 754.81,A -85,B 0,C 180,E1 2132.973,E2 2132.973} C_VEL
LIN {X 0,Y 571.072,Z 754.81,A -85,B 0,C 180,E1 2140.629,E2 2140.629} C_VEL
LIN {X 0,Y 571.044,Z 754.81,A -85,B 0,C 180,E1 2148.505,E2 2148.505} C_VEL
LIN {X 0,Y 570.91,Z 754.81,A -85,B 0,C 180,E1 2156.192,E2 2156.192} C_VEL
LIN {X 0,Y 570.802,Z 754.81,A -85,B 0,C 180,E1 2163.813,E2 2163.813} C_VEL
LIN {X 0,Y 570.675,Z 754.81,A -85,B 0,C 180,E1 2171.506,E2 2171.506} C_VEL
LIN {X 0,Y 570.582,Z 754.81,A -85,B 0,C 180,E1 2179.42,E2 2179.42} C_VEL
LIN {X 0,Y 570.406,Z 754.81,A -85,B 0,C 180,E1 2186.965,E2 2186.965} C_VEL
LIN {X 0,Y 570.387,Z 754.81,A -85,B 0,C 180,E1 2193.06,E2 2193.06} C_VEL
LIN {X 0,Y 570.639,Z 754.81,A -85,B 0,C 180,E1 2200.717,E2 2200.717} C_VEL
LIN {X 0,Y 570.612,Z 754.81,A -85,B 0,C 180,E1 2209.338,E2 2209.338} C_VEL
LIN {X 0,Y 570.562,Z 754.81,A -85,B 0,C 180,E1 2218.757,E2 2218.757} C_VEL
LIN {X 0,Y 570.412,Z 754.81,A -85,B 0,C 180,E1 2226.619,E2 2226.619} C_VEL
LIN {X 0,Y 570.821,Z 754.81,A -85,B 0,C 180,E1 2235.37,E2 2235.37} C_VEL
LIN {X 0,Y 571.111,Z 754.81,A -85,B 0,C 180,E1 2243.132,E2 2243.132} C_VEL
LIN {X 0,Y 570.548,Z 754.81,A -85,B 0,C 180,E1 2250.762,E2 2250.762} C_VEL
LIN {X 0,Y 571.419,Z 756.475,A -85,B 0,C 180,E1 2257.247,E2 2257.247} C_VEL
LIN {X 0,Y 572.343,Z 797.172,A -85,B 0,C 180,E1 2259.25,E2 2259.25} C_VEL
LIN {X 0,Y 571.948,Z 828.469,A -85,B 0,C 180,E1 2262.449,E2 2262.449} C_VEL
LIN {X 0,Y 571.704,Z 846.438,A -85,B 0,C 180,E1 2266.183,E2 2266.183} C_VEL
LIN {X 0,Y 571.416,Z 851.898,A -85,B 0,C 180,E1 2269.468,E2 2269.468} C_VEL
LIN {X 0,Y 571.748,Z 846.55,A -85,B 0,C 180,E1 2273.689,E2 2273.689} C_VEL
LIN {X 0,Y 571.941,Z 827.034,A -85,B 0,C 180,E1 2277.667,E2 2277.667} C_VEL
LIN {X 0,Y 572.31,Z 795.674,A -85,B 0,C 180,E1 2280.766,E2 2280.766} C_VEL
LIN {X 0,Y 571.173,Z 754.81,A -85,B 0,C 180,E1 2282.838,E2 2282.838} C_VEL
LIN {X 0,Y 570.712,Z 754.81,A -85,B 0,C 180,E1 2290.724,E2 2290.724} C_VEL
LIN {X 0,Y 570.655,Z 754.81,A -85,B 0,C 180,E1 2299.34,E2 2299.34} C_VEL
LIN {X 0,Y 570.606,Z 754.81,A -85,B 0,C 180,E1 2308.759,E2 2308.759} C_VEL
LIN {X 0,Y 570.459,Z 754.81,A -85,B 0,C 180,E1 2316.604,E2 2316.604} C_VEL
LIN {X 0,Y 570.794,Z 754.81,A -85,B 0,C 180,E1 2325.368,E2 2325.368} C_VEL
LIN {X 0,Y 571.081,Z 754.81,A -85,B 0,C 180,E1 2333.13,E2 2333.13} C_VEL
LIN {X 0,Y 570.968,Z 754.81,A -85,B 0,C 180,E1 2340.76,E2 2340.76} C_VEL
LIN {X 0,Y 570.75,Z 754.81,A -85,B 0,C 180,E1 2348.407,E2 2348.407} C_VEL
LIN {X 0,Y 571.03,Z 754.81,A -85,B 0,C 180,E1 2354.284,E2 2354.284} C_VEL
LIN {X 0,Y 562.66,Z 754.81,A -85,B 0,C 180,E1 2357.776,E2 2357.776} C_VEL
LIN {X 0,Y 562.766,Z 754.81,A -85,B 0,C 180,E1 2366.417,E2 2366.417} C_VEL
LIN {X 0,Y 562.845,Z 754.81,A -85,B 0,C 180,E1 2375.426,E2 2375.426} C_VEL
LIN {X 0,Y 562.718,Z 754.81,A -85,B 0,C 180,E1 2385.612,E2 2385.612} C_VEL
LIN {X 0,Y 562.597,Z 754.81,A -85,B 0,C 180,E1 2394.554,E2 2394.554} C_VEL
LIN {X 0,Y 562.777,Z 754.81,A -85,B 0,C 180,E1 2403.581,E2 2403.581} C_VEL
LIN {X 0,Y 563.179,Z 756.373,A -85,B 0,C 180,E1 2407.16,E2 2407.16} C_VEL
LIN {X 0,Y 566.618,Z 779.164,A -85,B 0,C 180,E1 2407.612,E2 2407.612} C_VEL
LIN {X 0,Y 566.48,Z 853.35,A -85,B 0,C 180,E1 2408.997,E2 2408.997} C_VEL
LIN {X 0,Y 565.455,Z 905.504,A -85,B 0,C 180,E1 2411.619,E2 2411.619} C_VEL
LIN {X 0,Y 564.444,Z 948.533,A -85,B 0,C 180,E1 2415.521,E2 2415.521} C_VEL
LIN {X 0,Y 563.695,Z 979.691,A -85,B 0,C 180,E1 2420.314,E2 2420.314} C_VEL
LIN {X 0,Y 563.373,Z 997.217,A -85,B 0,C 180,E1 2425.448,E2 2425.448} C_VEL
LIN {X 0,Y 563.256,Z 1001.838,A -85,B 0,C 180,E1 2430.772,E2 2430.772} C_VEL
LIN {X 0,Y 563.122,Z 993.116,A -85,B 0,C 180,E1 2436.189,E2 2436.189} C_VEL
LIN {X 0,Y 563.59,Z 970.846,A -85,B 0,C 180,E1 2441.348,E2 2441.348} C_VEL
LIN {X 0,Y 564.499,Z 934.483,A -85,B 0,C 180,E1 2445.996,E2 2445.996} C_VEL
LIN {X 0,Y 565.86,Z 887.667,A -85,B 0,C 180,E1 2449.486,E2 2449.486} C_VEL
LIN {X 0,Y 566.87,Z 835.594,A -85,B 0,C 180,E1 2451.506,E2 2451.506} C_VEL
LIN {X 0,Y 564.298,Z 759.079,A -85,B 0,C 180,E1 2452.756,E2 2452.756} C_VEL
LIN {X 0,Y 563.087,Z 754.81,A -85,B 0,C 180,E1 2453.004,E2 2453.004} C_VEL
LIN {X 0,Y 562.351,Z 754.81,A -85,B 0,C 180,E1 2461.786,E2 2461.786} C_VEL
LIN {X 0,Y 562.437,Z 754.81,A -85,B 0,C 180,E1 2469.741,E2 2469.741} C_VEL
LIN {X 0,Y 562.305,Z 754.81,A -85,B 0,C 180,E1 2477.918,E2 2477.918} C_VEL
LIN {X 0,Y 562.359,Z 754.81,A -85,B 0,C 180,E1 2485.394,E2 2485.394} C_VEL
LIN {X 0,Y 562.536,Z 754.81,A -85,B 0,C 180,E1 2493.571,E2 2493.571} C_VEL
LIN {X 0,Y 562.741,Z 754.81,A -85,B 0,C 180,E1 2501.936,E2 2501.936} C_VEL
LIN {X 0,Y 562.737,Z 754.81,A -85,B 0,C 180,E1 2509.907,E2 2509.907} C_VEL
LIN {X 0,Y 562.75,Z 754.81,A -85,B 0,C 180,E1 2517.684,E2 2517.684} C_VEL
LIN {X 0,Y 562.809,Z 754.81,A -85,B 0,C 180,E1 2523.867,E2 2523.867} C_VEL
LIN {X 0,Y 562.671,Z 754.81,A -85,B 0,C 180,E1 2531.672,E2 2531.672} C_VEL
LIN {X 0,Y 562.593,Z 754.81,A -85,B 0,C 180,E1 2539.707,E2 2539.707} C_VEL
LIN {X 0,Y 562.535,Z 754.81,A -85,B 0,C 180,E1 2548.173,E2 2548.173} C_VEL
LIN {X 0,Y 562.428,Z 754.81,A -85,B 0,C 180,E1 2557.382,E2 2557.382} C_VEL
LIN {X 0,Y 562.719,Z 754.81,A -85,B 0,C 180,E1 2566.551,E2 2566.551} C_VEL
LIN {X 0,Y 562.753,Z 754.81,A -85,B 0,C 180,E1 2576.439,E2 2576.439} C_VEL
LIN {X 0,Y 562.776,Z 754.81,A -85,B 0,C 180,E1 2585.293,E2 2585.293} C_VEL
LIN {X 0,Y 562.84,Z 754.81,A -85,B 0,C 180,E1 2595.158,E2 2595.158} C_VEL
LIN {X 0,Y 563.121,Z 754.81,A -85,B 0,C 180,E1 2603.034,E2 2603.034} C_VEL
LIN {X 0,Y 562.561,Z 754.81,A -85,B 0,C 180,E1 2610.772,E2 2610.772} C_VEL
LIN {X 0,Y 563.285,Z 756.48,A -85,B 0,C 180,E1 2617.06,E2 2617.06} C_VEL
LIN {X 0,Y 564.443,Z 795.657,A -85,B 0,C 180,E1 2618.99,E2 2618.99} C_VEL
LIN {X 0,Y 564.013,Z 827.711,A -85,B 0,C 180,E1 2622.233,E2 2622.233} C_VEL
LIN {X 0,Y 563.608,Z 847.293,A -85,B 0,C 180,E1 2626.422,E2 2626.422} C_VEL
LIN {X 0,Y 563.407,Z 851.946,A -85,B 0,C 180,E1 2629.675,E2 2629.675} C_VEL
LIN {X 0,Y 563.703,Z 845.64,A -85,B 0,C 180,E1 2634.048,E2 2634.048} C_VEL
LIN {X 0,Y 563.967,Z 824.705,A -85,B 0,C 180,E1 2638.093,E2 2638.093} C_VEL
LIN {X 0,Y 564.484,Z 791.607,A -85,B 0,C 180,E1 2641.198,E2 2641.198} C_VEL
LIN {X 0,Y 563.089,Z 754.81,A -85,B 0,C 180,E1 2643.016,E2 2643.016} C_VEL
LIN {X 0,Y 562.38,Z 754.81,A -85,B 0,C 180,E1 2652.089,E2 2652.089} C_VEL
LIN {X 0,Y 562.348,Z 754.81,A -85,B 0,C 180,E1 2660.274,E2 2660.274} C_VEL
LIN {X 0,Y 562.624,Z 754.81,A -85,B 0,C 180,E1 2668.264,E2 2668.264} C_VEL
LIN {X 0,Y 562.335,Z 754.81,A -85,B 0,C 180,E1 2676.962,E2 2676.962} C_VEL
LIN {X 0,Y 562.813,Z 754.81,A -85,B 0,C 180,E1 2685.156,E2 2685.156} C_VEL
LIN {X 0,Y 563.09,Z 754.81,A -85,B 0,C 180,E1 2693.032,E2 2693.032} C_VEL
LIN {X 0,Y 562.97,Z 754.81,A -85,B 0,C 180,E1 2700.77,E2 2700.77} C_VEL
LIN {X 0,Y 562.73,Z 754.81,A -85,B 0,C 180,E1 2708.528,E2 2708.528} C_VEL
LIN {X 0,Y 562.572,Z 754.81,A -85,B 0,C 180,E1 2716.452,E2 2716.452} C_VEL
LIN {X 0,Y 562.66,Z 754.81,A -85,B 0,C 180,E1 2717.776,E2 2717.776} C_VEL
LIN {X 0,Y 554.867,Z 754.81,A -85,B 0,C 180,E1 2721.344,E2 2721.344} C_VEL
LIN {X 0,Y 554.56,Z 754.81,A -85,B 0,C 180,E1 2730.458,E2 2730.458} C_VEL
LIN {X 0,Y 554.545,Z 754.81,A -85,B 0,C 180,E1 2738.746,E2 2738.746} C_VEL
LIN {X 0,Y 554.558,Z 754.81,A -85,B 0,C 180,E1 2746.48,E2 2746.48} C_VEL
LIN {X 0,Y 554.625,Z 754.81,A -85,B 0,C 180,E1 2753.965,E2 2753.965} C_VEL
LIN {X 0,Y 554.78,Z 754.81,A -85,B 0,C 180,E1 2763.17,E2 2763.17} C_VEL
LIN {X 0,Y 555.082,Z 756.43,A -85,B 0,C 180,E1 2766.808,E2 2766.808} C_VEL
LIN {X 0,Y 559.234,Z 779.164,A -85,B 0,C 180,E1 2767.301,E2 2767.301} C_VEL
LIN {X 0,Y 559.012,Z 852.28,A -85,B 0,C 180,E1 2768.665,E2 2768.665} C_VEL
LIN {X 0,Y 557.83,Z 904.011,A -85,B 0,C 180,E1 2771.255,E2 2771.255} C_VEL
LIN {X 0,Y 556.694,Z 947.128,A -85,B 0,C 180,E1 2775.151,E2 2775.151} C_VEL
LIN {X 0,Y 555.759,Z 979.691,A -85,B 0,C 180,E1 2780.174,E2 2780.174} C_VEL
LIN {X 0,Y 555.425,Z 997.049,A -85,B 0,C 180,E1 2785.299,E2 2785.299} C_VEL
LIN {X 0,Y 555.252,Z 1001.838,A -85,B 0,C 180,E1 2790.784,E2 2790.784} C_VEL
LIN {X 0,Y 555.244,Z 994.252,A -85,B 0,C 180,E1 2795.883,E2 2795.883} C_VEL
LIN {X 0,Y 555.638,Z 973.17,A -85,B 0,C 180,E1 2801.095,E2 2801.095} C_VEL
LIN {X 0,Y 556.683,Z 938.395,A -85,B 0,C 180,E1 2805.82,E2 2805.82} C_VEL
LIN {X 0,Y 558.156,Z 892.871,A -85,B 0,C 180,E1 2809.456,E2 2809.456} C_VEL
LIN {X 0,Y 559.352,Z 840.842,A -85,B 0,C 180,E1 2811.671,E2 2811.671} C_VEL
LIN {X 0,Y 557.286,Z 762.087,A -85,B 0,C 180,E1 2813.017,E2 2813.017} C_VEL
LIN {X 0,Y 554.996,Z 754.81,A -85,B 0,C 180,E1 2813.359,E2 2813.359} C_VEL
LIN {X 0,Y 554.349,Z 754.81,A -85,B 0,C 180,E1 2822.265,E2 2822.265} C_VEL
LIN {X 0,Y 554.409,Z 754.81,A -85,B 0,C 180,E1 2830.036,E2 2830.036} C_VEL
LIN {X 0,Y 554.327,Z 754.81,A -85,B 0,C 180,E1 2837.88,E2 2837.88} C_VEL
LIN {X 0,Y 554.263,Z 754.81,A -85,B 0,C 180,E1 2845.858,E2 2845.858} C_VEL
LIN {X 0,Y 554.561,Z 754.81,A -85,B 0,C 180,E1 2853.161,E2 2853.161} C_VEL
LIN {X 0,Y 554.76,Z 754.81,A -85,B 0,C 180,E1 2861.666,E2 2861.666} C_VEL
LIN {X 0,Y 554.796,Z 754.81,A -85,B 0,C 180,E1 2869.761,E2 2869.761} C_VEL
LIN {X 0,Y 554.751,Z 754.81,A -85,B 0,C 180,E1 2877.65,E2 2877.65} C_VEL
LIN {X 0,Y 554.818,Z 754.81,A -85,B 0,C 180,E1 2883.923,E2 2883.923} C_VEL
LIN {X 0,Y 554.672,Z 754.81,A -85,B 0,C 180,E1 2891.843,E2 2891.843} C_VEL
LIN {X 0,Y 554.626,Z 754.81,A -85,B 0,C 180,E1 2900.002,E2 2900.002} C_VEL
LIN {X 0,Y 554.617,Z 754.81,A -85,B 0,C 180,E1 2908.612,E2 2908.612} C_VEL
LIN {X 0,Y 554.522,Z 754.81,A -85,B 0,C 180,E1 2918.742,E2 2918.742} C_VEL
LIN {X 0,Y 554.616,Z 754.81,A -85,B 0,C 180,E1 2928.807,E2 2928.807} C_VEL
LIN {X 0,Y 554.608,Z 754.81,A -85,B 0,C 180,E1 2937.752,E2 2937.752} C_VEL
LIN {X 0,Y 554.355,Z 754.81,A -85,B 0,C 180,E1 2946.612,E2 2946.612} C_VEL
LIN {X 0,Y 554.844,Z 754.81,A -85,B 0,C 180,E1 2954.939,E2 2954.939} C_VEL
LIN {X 0,Y 555.135,Z 754.81,A -85,B 0,C 180,E1 2962.933,E2 2962.933} C_VEL
LIN {X 0,Y 554.548,Z 754.81,A -85,B 0,C 180,E1 2970.783,E2 2970.783} C_VEL
LIN {X 0,Y 555.152,Z 756.49,A -85,B 0,C 180,E1 2976.868,E2 2976.868} C_VEL
LIN {X 0,Y 556.576,Z 795.498,A -85,B 0,C 180,E1 2978.822,E2 2978.822} C_VEL
LIN {X 0,Y 556.075,Z 826.956,A -85,B 0,C 180,E1 2982.01,E2 2982.01} C_VEL
LIN {X 0,Y 555.755,Z 845.767,A -85,B 0,C 180,E1 2985.846,E2 2985.846} C_VEL
LIN {X 0,Y 555.375,Z 851.998,A -85,B 0,C 180,E1 2989.972,E2 2989.972} C_VEL
LIN {X 0,Y 555.638,Z 844.694,A -85,B 0,C 180,E1 2994.391,E2 2994.391} C_VEL
LIN {X 0,Y 555.966,Z 823.34,A -85,B 0,C 180,E1 2998.394,E2 2998.394} C_VEL
LIN {X 0,Y 556.574,Z 789.436,A -85,B 0,C 180,E1 3001.501,E2 3001.501} C_VEL
LIN {X 0,Y 554.986,Z 754.81,A -85,B 0,C 180,E1 3003.263,E2 3003.263} C_VEL
LIN {X 0,Y 554.386,Z 754.81,A -85,B 0,C 180,E1 3012.118,E2 3012.118} C_VEL
LIN {X 0,Y 554.396,Z 754.81,A -85,B 0,C 180,E1 3019.962,E2 3019.962} C_VEL
LIN {X 0,Y 554.649,Z 754.81,A -85,B 0,C 180,E1 3027.753,E2 3027.753} C_VEL
LIN {X 0,Y 554.397,Z 754.81,A -85,B 0,C 180,E1 3036.613,E2 3036.613} C_VEL
LIN {X 0,Y 554.818,Z 754.81,A -85,B 0,C 180,E1 3044.937,E2 3044.937} C_VEL
LIN {X 0,Y 555.105,Z 754.81,A -85,B 0,C 180,E1 3052.932,E2 3052.932} C_VEL
LIN {X 0,Y 554.965,Z 754.81,A -85,B 0,C 180,E1 3060.781,E2 3060.781} C_VEL
LIN {X 0,Y 554.744,Z 754.81,A -85,B 0,C 180,E1 3068.651,E2 3068.651} C_VEL
LIN {X 0,Y 554.573,Z 754.81,A -85,B 0,C 180,E1 3076.696,E2 3076.696} C_VEL
LIN {X 0,Y 554.867,Z 754.81,A -85,B 0,C 180,E1 3081.344,E2 3081.344} C_VEL
LIN {X 0,Y 546.459,Z 754.81,A -85,B 0,C 180,E1 3084.937,E2 3084.937} C_VEL
LIN {X 0,Y 546.376,Z 754.81,A -85,B 0,C 180,E1 3092.791,E2 3092.791} C_VEL
LIN {X 0,Y 546.446,Z 754.81,A -85,B 0,C 180,E1 3100.737,E2 3100.737} C_VEL
LIN {X 0,Y 546.446,Z 754.81,A -85,B 0,C 180,E1 3109.789,E2 3109.789} C_VEL
LIN {X 0,Y 546.517,Z 754.81,A -85,B 0,C 180,E1 3119.089,E2 3119.089} C_VEL
LIN {X 0,Y 546.929,Z 755.828,A -85,B 0,C 180,E1 3126.433,E2 3126.433} C_VEL
LIN {X 0,Y 551.837,Z 778.529,A -85,B 0,C 180,E1 3126.97,E2 3126.97} C_VEL
LIN {X 0,Y 551.548,Z 852.489,A -85,B 0,C 180,E1 3128.369,E2 3128.369} C_VEL
LIN {X 0,Y 550.166,Z 904.014,A -85,B 0,C 180,E1 3130.984,E2 3130.984} C_VEL
LIN {X 0,Y 548.883,Z 946.744,A -85,B 0,C 180,E1 3134.89,E2 3134.89} C_VEL
LIN {X 0,Y 548.034,Z 977.737,A -85,B 0,C 180,E1 3139.631,E2 3139.631} C_VEL
LIN {X 0,Y 547.447,Z 997.048,A -85,B 0,C 180,E1 3145.23,E2 3145.23} C_VEL
LIN {X 0,Y 547.276,Z 1001.837,A -85,B 0,C 180,E1 3150.795,E2 3150.795} C_VEL
LIN {X 0,Y 547.229,Z 994.252,A -85,B 0,C 180,E1 3155.97,E2 3155.97} C_VEL
LIN {X 0,Y 547.68,Z 972.801,A -85,B 0,C 180,E1 3161.326,E2 3161.326} C_VEL
LIN {X 0,Y 548.855,Z 938.394,A -85,B 0,C 180,E1 3166.052,E2 3166.052} C_VEL
LIN {X 0,Y 550.539,Z 892.868,A -85,B 0,C 180,E1 3169.736,E2 3169.736} C_VEL
LIN {X 0,Y 551.928,Z 840.42,A -85,B 0,C 180,E1 3171.989,E2 3171.989} C_VEL
LIN {X 0,Y 549.822,Z 763.898,A -85,B 0,C 180,E1 3173.323,E2 3173.323} C_VEL
LIN {X 0,Y 546.961,Z 754.81,A -85,B 0,C 180,E1 3173.723,E2 3173.723} C_VEL
LIN {X 0,Y 546.375,Z 754.81,A -85,B 0,C 180,E1 3182.795,E2 3182.795} C_VEL
LIN {X 0,Y 546.413,Z 754.81,A -85,B 0,C 180,E1 3190.744,E2 3190.744} C_VEL
LIN {X 0,Y 546.369,Z 754.81,A -85,B 0,C 180,E1 3199.804,E2 3199.804} C_VEL
LIN {X 0,Y 546.452,Z 754.81,A -85,B 0,C 180,E1 3209.088,E2 3209.088} C_VEL
LIN {X 0,Y 546.815,Z 754.81,A -85,B 0,C 180,E1 3218.393,E2 3218.393} C_VEL
LIN {X 0,Y 547.056,Z 754.81,A -85,B 0,C 180,E1 3227.994,E2 3227.994} C_VEL
LIN {X 0,Y 546.959,Z 754.81,A -85,B 0,C 180,E1 3236.025,E2 3236.025} C_VEL
LIN {X 0,Y 546.81,Z 754.81,A -85,B 0,C 180,E1 3243.981,E2 3243.981} C_VEL
LIN {X 0,Y 546.674,Z 754.81,A -85,B 0,C 180,E1 3252.019,E2 3252.019} C_VEL
LIN {X 0,Y 546.641,Z 754.81,A -85,B 0,C 180,E1 3260.307,E2 3260.307} C_VEL
LIN {X 0,Y 546.61,Z 754.81,A -85,B 0,C 180,E1 3269.07,E2 3269.07} C_VEL
LIN {X 0,Y 546.527,Z 754.81,A -85,B 0,C 180,E1 3278.667,E2 3278.667} C_VEL
LIN {X 0,Y 546.729,Z 754.81,A -85,B 0,C 180,E1 3287.357,E2 3287.357} C_VEL
LIN {X 0,Y 546.602,Z 754.81,A -85,B 0,C 180,E1 3297.867,E2 3297.867} C_VEL
LIN {X 0,Y 546.454,Z 754.81,A -85,B 0,C 180,E1 3306.253,E2 3306.253} C_VEL
LIN {X 0,Y 546.839,Z 754.81,A -85,B 0,C 180,E1 3314.713,E2 3314.713} C_VEL
LIN {X 0,Y 547.137,Z 754.81,A -85,B 0,C 180,E1 3322.829,E2 3322.829} C_VEL
LIN {X 0,Y 546.546,Z 754.81,A -85,B 0,C 180,E1 3330.795,E2 3330.795} C_VEL
LIN {X 0,Y 547.06,Z 756.46,A -85,B 0,C 180,E1 3336.67,E2 3336.67} C_VEL
LIN {X 0,Y 548.706,Z 792.561,A -85,B 0,C 180,E1 3338.449,E2 3338.449} C_VEL
LIN {X 0,Y 548.08,Z 824.737,A -85,B 0,C 180,E1 3341.585,E2 3341.585} C_VEL
LIN {X 0,Y 547.774,Z 845.416,A -85,B 0,C 180,E1 3345.671,E2 3345.671} C_VEL
LIN {X 0,Y 547.333,Z 851.937,A -85,B 0,C 180,E1 3350.278,E2 3350.278} C_VEL
LIN {X 0,Y 547.521,Z 843.477,A -85,B 0,C 180,E1 3354.815,E2 3354.815} C_VEL
LIN {X 0,Y 548.01,Z 820.683,A -85,B 0,C 180,E1 3358.854,E2 3358.854} C_VEL
LIN {X 0,Y 548.757,Z 785.558,A -85,B 0,C 180,E1 3361.91,E2 3361.91} C_VEL
LIN {X 0,Y 546.925,Z 754.81,A -85,B 0,C 180,E1 3363.404,E2 3363.404} C_VEL
LIN {X 0,Y 546.314,Z 754.81,A -85,B 0,C 180,E1 3372.888,E2 3372.888} C_VEL
LIN {X 0,Y 546.43,Z 754.81,A -85,B 0,C 180,E1 3379.795,E2 3379.795} C_VEL
LIN {X 0,Y 546.462,Z 754.81,A -85,B 0,C 180,E1 3389.084,E2 3389.084} C_VEL
LIN {X 0,Y 546.496,Z 754.81,A -85,B 0,C 180,E1 3396.254,E2 3396.254} C_VEL
LIN {X 0,Y 546.814,Z 754.81,A -85,B 0,C 180,E1 3404.711,E2 3404.711} C_VEL
LIN {X 0,Y 547.103,Z 754.81,A -85,B 0,C 180,E1 3412.828,E2 3412.828} C_VEL
LIN {X 0,Y 546.975,Z 754.81,A -85,B 0,C 180,E1 3420.793,E2 3420.793} C_VEL
LIN {X 0,Y 546.729,Z 754.81,A -85,B 0,C 180,E1 3428.779,E2 3428.779} C_VEL
LIN {X 0,Y 546.58,Z 754.81,A -85,B 0,C 180,E1 3436.947,E2 3436.947} C_VEL
LIN {X 0,Y 546.459,Z 754.81,A -85,B 0,C 180,E1 3444.937,E2 3444.937} C_VEL
LIN {X 0,Y 538.643,Z 754.81,A -85,B 0,C 180,E1 3448.605,E2 3448.605} C_VEL
LIN {X 0,Y 538.684,Z 754.81,A -85,B 0,C 180,E1 3457.276,E2 3457.276} C_VEL
LIN {X 0,Y 538.475,Z 754.81,A -85,B 0,C 180,E1 3466.333,E2 3466.333} C_VEL
LIN {X 0,Y 538.423,Z 754.81,A -85,B 0,C 180,E1 3474.704,E2 3474.704} C_VEL
LIN {X 0,Y 538.698,Z 754.81,A -85,B 0,C 180,E1 3484.11,E2 3484.11} C_VEL
LIN {X 0,Y 538.913,Z 756.115,A -85,B 0,C 180,E1 3486.065,E2 3486.065} C_VEL
LIN {X 0,Y 544.488,Z 779.281,A -85,B 0,C 180,E1 3486.652,E2 3486.652} C_VEL
LIN {X 0,Y 544.071,Z 853.425,A -85,B 0,C 180,E1 3488.091,E2 3488.091} C_VEL
LIN {X 0,Y 542.498,Z 905.497,A -85,B 0,C 180,E1 3490.811,E2 3490.811} C_VEL
LIN {X 0,Y 540.998,Z 948.305,A -85,B 0,C 180,E1 3494.85,E2 3494.85} C_VEL
LIN {X 0,Y 539.959,Z 979.69,A -85,B 0,C 180,E1 3499.884,E2 3499.884} C_VEL
LIN {X 0,Y 539.478,Z 997.048,A -85,B 0,C 180,E1 3505.159,E2 3505.159} C_VEL
LIN {X 0,Y 539.272,Z 1001.837,A -85,B 0,C 180,E1 3510.807,E2 3510.807} C_VEL
LIN {X 0,Y 539.208,Z 994.252,A -85,B 0,C 180,E1 3516.059,E2 3516.059} C_VEL
LIN {X 0,Y 539.733,Z 972.474,A -85,B 0,C 180,E1 3521.557,E2 3521.557} C_VEL
LIN {X 0,Y 541.027,Z 938.393,A -85,B 0,C 180,E1 3526.291,E2 3526.291} C_VEL
LIN {X 0,Y 542.951,Z 892.866,A -85,B 0,C 180,E1 3530.023,E2 3530.023} C_VEL
LIN {X 0,Y 544.508,Z 840.419,A -85,B 0,C 180,E1 3532.305,E2 3532.305} C_VEL
LIN {X 0,Y 542.425,Z 765.527,A -85,B 0,C 180,E1 3533.637,E2 3533.637} C_VEL
LIN {X 0,Y 538.893,Z 754.81,A -85,B 0,C 180,E1 3534.101,E2 3534.101} C_VEL
LIN {X 0,Y 538.418,Z 754.81,A -85,B 0,C 180,E1 3543.754,E2 3543.754} C_VEL
LIN {X 0,Y 538.434,Z 754.81,A -85,B 0,C 180,E1 3551.682,E2 3551.682} C_VEL
LIN {X 0,Y 538.464,Z 754.81,A -85,B 0,C 180,E1 3560.81,E2 3560.81} C_VEL
LIN {X 0,Y 538.617,Z 754.81,A -85,B 0,C 180,E1 3570.46,E2 3570.46} C_VEL
LIN {X 0,Y 538.792,Z 754.81,A -85,B 0,C 180,E1 3581.103,E2 3581.103} C_VEL
LIN {X 0,Y 538.81,Z 754.81,A -85,B 0,C 180,E1 3589.453,E2 3589.453} C_VEL
LIN {X 0,Y 538.781,Z 754.81,A -85,B 0,C 180,E1 3597.581,E2 3597.581} C_VEL
LIN {X 0,Y 538.826,Z 754.81,A -85,B 0,C 180,E1 3604.04,E2 3604.04} C_VEL
LIN {X 0,Y 538.682,Z 754.81,A -85,B 0,C 180,E1 3612.2,E2 3612.2} C_VEL
LIN {X 0,Y 538.677,Z 754.81,A -85,B 0,C 180,E1 3620.621,E2 3620.621} C_VEL
LIN {X 0,Y 538.581,Z 754.81,A -85,B 0,C 180,E1 3629.546,E2 3629.546} C_VEL
LIN {X 0,Y 538.514,Z 754.81,A -85,B 0,C 180,E1 3639.353,E2 3639.353} C_VEL
LIN {X 0,Y 538.518,Z 754.81,A -85,B 0,C 180,E1 3648.528,E2 3648.528} C_VEL
LIN {X 0,Y 538.444,Z 754.81,A -85,B 0,C 180,E1 3658.572,E2 3658.572} C_VEL
LIN {X 0,Y 538.42,Z 754.81,A -85,B 0,C 180,E1 3666.356,E2 3666.356} C_VEL
LIN {X 0,Y 538.829,Z 754.81,A -85,B 0,C 180,E1 3674.48,E2 3674.48} C_VEL
LIN {X 0,Y 539.133,Z 754.81,A -85,B 0,C 180,E1 3682.722,E2 3682.722} C_VEL
LIN {X 0,Y 538.54,Z 754.81,A -85,B 0,C 180,E1 3690.807,E2 3690.807} C_VEL
LIN {X 0,Y 538.906,Z 756.373,A -85,B 0,C 180,E1 3696.463,E2 3696.463} C_VEL
LIN {X 0,Y 540.951,Z 787.783,A -85,B 0,C 180,E1 3697.961,E2 3697.961} C_VEL
LIN {X 0,Y 540.161,Z 820.727,A -85,B 0,C 180,E1 3700.931,E2 3700.931} C_VEL
LIN {X 0,Y 539.683,Z 843.683,A -85,B 0,C 180,E1 3705.083,E2 3705.083} C_VEL
LIN {X 0,Y 539.301,Z 851.908,A -85,B 0,C 180,E1 3709.49,E2 3709.49} C_VEL
LIN {X 0,Y 539.68,Z 846.12,A -85,B 0,C 180,E1 3714.062,E2 3714.062} C_VEL
LIN {X 0,Y 540.052,Z 825.598,A -85,B 0,C 180,E1 3718.331,E2 3718.331} C_VEL
LIN {X 0,Y 540.83,Z 793.116,A -85,B 0,C 180,E1 3721.591,E2 3721.591} C_VEL
LIN {X 0,Y 539.281,Z 757.164,A -85,B 0,C 180,E1 3723.413,E2 3723.413} C_VEL
LIN {X 0,Y 538.821,Z 754.81,A -85,B 0,C 180,E1 3723.811,E2 3723.811} C_VEL
LIN {X 0,Y 538.397,Z 754.81,A -85,B 0,C 180,E1 3731.671,E2 3731.671} C_VEL
LIN {X 0,Y 538.223,Z 754.81,A -85,B 0,C 180,E1 3740.84,E2 3740.84} C_VEL
LIN {X 0,Y 538.428,Z 754.81,A -85,B 0,C 180,E1 3749.276,E2 3749.276} C_VEL
LIN {X 0,Y 538.118,Z 754.81,A -85,B 0,C 180,E1 3757.62,E2 3757.62} C_VEL
LIN {X 0,Y 538.511,Z 754.81,A -85,B 0,C 180,E1 3766.467,E2 3766.467} C_VEL
LIN {X 0,Y 538.83,Z 754.81,A -85,B 0,C 180,E1 3774.341,E2 3774.341} C_VEL
LIN {X 0,Y 538.88,Z 754.81,A -85,B 0,C 180,E1 3781.331,E2 3781.331} C_VEL
LIN {X 0,Y 538.737,Z 754.81,A -85,B 0,C 180,E1 3788.911,E2 3788.911} C_VEL
LIN {X 0,Y 538.583,Z 754.81,A -85,B 0,C 180,E1 3797.207,E2 3797.207} C_VEL
LIN {X 0,Y 538.582,Z 754.81,A -85,B 0,C 180,E1 3805.894,E2 3805.894} C_VEL
LIN {X 0,Y 538.643,Z 754.81,A -85,B 0,C 180,E1 3808.605,E2 3808.605} C_VEL
LIN {X 0,Y 530.32,Z 754.81,A -85,B 0,C 180,E1 3812.295,E2 3812.295} C_VEL
LIN {X 0,Y 530.4,Z 754.81,A -85,B 0,C 180,E1 3820.694,E2 3820.694} C_VEL
LIN {X 0,Y 530.363,Z 754.81,A -85,B 0,C 180,E1 3829.924,E2 3829.924} C_VEL
LIN {X 0,Y 530.284,Z 754.81,A -85,B 0,C 180,E1 3838.033,E2 3838.033} C_VEL
LIN {X 0,Y 531.002,Z 756.76,A -85,B 0,C 180,E1 3845.743,E2 3845.743} C_VEL
LIN {X 0,Y 537.171,Z 780.676,A -85,B 0,C 180,E1 3846.334,E2 3846.334} C_VEL
LIN {X 0,Y 536.633,Z 853.549,A -85,B 0,C 180,E1 3847.776,E2 3847.776} C_VEL
LIN {X 0,Y 534.849,Z 905.495,A -85,B 0,C 180,E1 3850.526,E2 3850.526} C_VEL
LIN {X 0,Y 533.207,Z 947.921,A -85,B 0,C 180,E1 3854.577,E2 3854.577} C_VEL
LIN {X 0,Y 532.035,Z 979.75,A -85,B 0,C 180,E1 3859.744,E2 3859.744} C_VEL
LIN {X 0,Y 531.507,Z 997.047,A -85,B 0,C 180,E1 3865.087,E2 3865.087} C_VEL
LIN {X 0,Y 531.28,Z 1001.837,A -85,B 0,C 180,E1 3870.819,E2 3870.819} C_VEL
LIN {X 0,Y 531.2,Z 994.252,A -85,B 0,C 180,E1 3876.151,E2 3876.151} C_VEL
LIN {X 0,Y 531.779,Z 973.564,A -85,B 0,C 180,E1 3881.524,E2 3881.524} C_VEL
LIN {X 0,Y 533.216,Z 940.315,A -85,B 0,C 180,E1 3886.323,E2 3886.323} C_VEL
LIN {X 0,Y 535.299,Z 894.571,A -85,B 0,C 180,E1 3890.214,E2 3890.214} C_VEL
LIN {X 0,Y 537.078,Z 842.574,A -85,B 0,C 180,E1 3892.57,E2 3892.57} C_VEL
LIN {X 0,Y 535.226,Z 767.806,A -85,B 0,C 180,E1 3893.941,E2 3893.941} C_VEL
LIN {X 0,Y 530.84,Z 754.81,A -85,B 0,C 180,E1 3894.49,E2 3894.49} C_VEL
LIN {X 0,Y 530.429,Z 754.81,A -85,B 0,C 180,E1 3903.911,E2 3903.911} C_VEL
LIN {X 0,Y 530.479,Z 754.81,A -85,B 0,C 180,E1 3913.16,E2 3913.16} C_VEL
LIN {X 0,Y 530.496,Z 754.81,A -85,B 0,C 180,E1 3922.048,E2 3922.048} C_VEL
LIN {X 0,Y 530.595,Z 754.81,A -85,B 0,C 180,E1 3931.844,E2 3931.844} C_VEL
LIN {X 0,Y 530.824,Z 754.81,A -85,B 0,C 180,E1 3940.808,E2 3940.808} C_VEL
LIN {X 0,Y 530.837,Z 754.81,A -85,B 0,C 180,E1 3949.293,E2 3949.293} C_VEL
LIN {X 0,Y 530.781,Z 754.81,A -85,B 0,C 180,E1 3957.544,E2 3957.544} C_VEL
LIN {X 0,Y 530.819,Z 754.81,A -85,B 0,C 180,E1 3964.101,E2 3964.101} C_VEL
LIN {X 0,Y 530.708,Z 754.81,A -85,B 0,C 180,E1 3972.386,E2 3972.386} C_VEL
LIN {X 0,Y 530.722,Z 754.81,A -85,B 0,C 180,E1 3981.669,E2 3981.669} C_VEL
LIN {X 0,Y 530.45,Z 754.81,A -85,B 0,C 180,E1 3991.958,E2 3991.958} C_VEL
LIN {X 0,Y 530.313,Z 754.81,A -85,B 0,C 180,E1 4000.681,E2 4000.681} C_VEL
LIN {X 0,Y 530.235,Z 754.81,A -85,B 0,C 180,E1 4009.911,E2 4009.911} C_VEL
LIN {X 0,Y 530.407,Z 754.81,A -85,B 0,C 180,E1 4018.04,E2 4018.04} C_VEL
LIN {X 0,Y 530.149,Z 754.81,A -85,B 0,C 180,E1 4027.266,E2 4027.266} C_VEL
LIN {X 0,Y 530.596,Z 754.81,A -85,B 0,C 180,E1 4035.929,E2 4035.929} C_VEL
LIN {X 0,Y 530.857,Z 754.81,A -85,B 0,C 180,E1 4044.257,E2 4044.257} C_VEL
LIN {X 0,Y 530.528,Z 754.81,A -85,B 0,C 180,E1 4050.819,E2 4050.819} C_VEL
LIN {X 0,Y 530.698,Z 755.816,A -85,B 0,C 180,E1 4056.207,E2 4056.207} C_VEL
LIN {X 0,Y 533.132,Z 785.936,A -85,B 0,C 180,E1 4057.667,E2 4057.667} C_VEL
LIN {X 0,Y 532.224,Z 819.833,A -85,B 0,C 180,E1 4060.68,E2 4060.68} C_VEL
LIN {X 0,Y 531.654,Z 843.243,A -85,B 0,C 180,E1 4064.886,E2 4064.886} C_VEL
LIN {X 0,Y 531.298,Z 851.784,A -85,B 0,C 180,E1 4069.176,E2 4069.176} C_VEL
LIN {X 0,Y 531.703,Z 846.607,A -85,B 0,C 180,E1 4073.951,E2 4073.951} C_VEL
LIN {X 0,Y 532.126,Z 827.439,A -85,B 0,C 180,E1 4078.186,E2 4078.186} C_VEL
LIN {X 0,Y 532.953,Z 795.949,A -85,B 0,C 180,E1 4081.554,E2 4081.554} C_VEL
LIN {X 0,Y 531.509,Z 758.448,A -85,B 0,C 180,E1 4083.591,E2 4083.591} C_VEL
LIN {X 0,Y 530.811,Z 754.81,A -85,B 0,C 180,E1 4083.882,E2 4083.882} C_VEL
LIN {X 0,Y 530.26,Z 754.81,A -85,B 0,C 180,E1 4093.129,E2 4093.129} C_VEL
LIN {X 0,Y 530.078,Z 754.81,A -85,B 0,C 180,E1 4102.008,E2 4102.008} C_VEL
LIN {X 0,Y 530.373,Z 754.81,A -85,B 0,C 180,E1 4110.774,E2 4110.774} C_VEL
LIN {X 0,Y 529.995,Z 754.81,A -85,B 0,C 180,E1 4119.026,E2 4119.026} C_VEL
LIN {X 0,Y 530.55,Z 754.81,A -85,B 0,C 180,E1 4125.927,E2 4125.927} C_VEL
LIN {X 0,Y 530.834,Z 754.81,A -85,B 0,C 180,E1 4134.255,E2 4134.255} C_VEL
LIN {X 0,Y 531.006,Z 754.81,A -85,B 0,C 180,E1 4140.817,E2 4140.817} C_VEL
LIN {X 0,Y 530.701,Z 754.81,A -85,B 0,C 180,E1 4149.411,E2 4149.411} C_VEL
LIN {X 0,Y 530.596,Z 754.81,A -85,B 0,C 180,E1 4157.474,E2 4157.474} C_VEL
LIN {X 0,Y 530.614,Z 754.81,A -85,B 0,C 180,E1 4166.312,E2 4166.312} C_VEL
LIN {X 0,Y 530.32,Z 754.81,A -85,B 0,C 180,E1 4172.295,E2 4172.295} C_VEL
LIN {X 0,Y 522.464,Z 754.81,A -85,B 0,C 180,E1 4176.074,E2 4176.074} C_VEL
LIN {X 0,Y 522.513,Z 754.81,A -85,B 0,C 180,E1 4185.359,E2 4185.359} C_VEL
LIN {X 0,Y 522.311,Z 754.81,A -85,B 0,C 180,E1 4195.489,E2 4195.489} C_VEL
LIN {X 0,Y 522.717,Z 754.81,A -85,B 0,C 180,E1 4205.37,E2 4205.37} C_VEL
LIN {X 0,Y 529.693,Z 781.291,A -85,B 0,C 180,E1 4206.037,E2 4206.037} C_VEL
LIN {X 0,Y 529.227,Z 853.487,A -85,B 0,C 180,E1 4207.448,E2 4207.448} C_VEL
LIN {X 0,Y 527.275,Z 904.434,A -85,B 0,C 180,E1 4210.155,E2 4210.155} C_VEL
LIN {X 0,Y 525.44,Z 947.494,A -85,B 0,C 180,E1 4214.291,E2 4214.291} C_VEL
LIN {X 0,Y 524.103,Z 979.749,A -85,B 0,C 180,E1 4219.587,E2 4219.587} C_VEL
LIN {X 0,Y 523.549,Z 997.047,A -85,B 0,C 180,E1 4225.012,E2 4225.012} C_VEL
LIN {X 0,Y 523.305,Z 1001.837,A -85,B 0,C 180,E1 4230.831,E2 4230.831} C_VEL
LIN {X 0,Y 523.211,Z 994.252,A -85,B 0,C 180,E1 4236.245,E2 4236.245} C_VEL
LIN {X 0,Y 523.82,Z 973.563,A -85,B 0,C 180,E1 4241.701,E2 4241.701} C_VEL
LIN {X 0,Y 525.373,Z 940.314,A -85,B 0,C 180,E1 4246.574,E2 4246.574} C_VEL
LIN {X 0,Y 527.715,Z 894.879,A -85,B 0,C 180,E1 4250.497,E2 4250.497} C_VEL
LIN {X 0,Y 529.675,Z 842.307,A -85,B 0,C 180,E1 4252.904,E2 4252.904} C_VEL
LIN {X 0,Y 527.577,Z 769.253,A -85,B 0,C 180,E1 4254.213,E2 4254.213} C_VEL
LIN {X 0,Y 522.839,Z 754.81,A -85,B 0,C 180,E1 4254.729,E2 4254.729} C_VEL
LIN {X 0,Y 522.486,Z 754.81,A -85,B 0,C 180,E1 4264.499,E2 4264.499} C_VEL
LIN {X 0,Y 522.508,Z 754.81,A -85,B 0,C 180,E1 4274.641,E2 4274.641} C_VEL
LIN {X 0,Y 522.4,Z 754.81,A -85,B 0,C 180,E1 4283.453,E2 4283.453} C_VEL
LIN {X 0,Y 522.403,Z 754.81,A -85,B 0,C 180,E1 4293.242,E2 4293.242} C_VEL
LIN {X 0,Y 522.632,Z 754.81,A -85,B 0,C 180,E1 4302.251,E2 4302.251} C_VEL
LIN {X 0,Y 522.752,Z 754.81,A -85,B 0,C 180,E1 4310.815,E2 4310.815} C_VEL
LIN {X 0,Y 523.021,Z 754.81,A -85,B 0,C 180,E1 4319.171,E2 4319.171} C_VEL
LIN {X 0,Y 523.168,Z 754.81,A -85,B 0,C 180,E1 4329.182,E2 4329.182} C_VEL
LIN {X 0,Y 522.773,Z 754.81,A -85,B 0,C 180,E1 4337.749,E2 4337.749} C_VEL
LIN {X 0,Y 522.406,Z 754.81,A -85,B 0,C 180,E1 4346.763,E2 4346.763} C_VEL
LIN {X 0,Y 522.112,Z 754.81,A -85,B 0,C 180,E1 4354.528,E2 4354.528} C_VEL
LIN {X 0,Y 522.179,Z 754.81,A -85,B 0,C 180,E1 4363.078,E2 4363.078} C_VEL
LIN {X 0,Y 522.052,Z 754.81,A -85,B 0,C 180,E1 4371.318,E2 4371.318} C_VEL
LIN {X 0,Y 522.268,Z 754.81,A -85,B 0,C 180,E1 4379.435,E2 4379.435} C_VEL
LIN {X 0,Y 522.176,Z 754.81,A -85,B 0,C 180,E1 4386.899,E2 4386.899} C_VEL
LIN {X 0,Y 522.613,Z 754.81,A -85,B 0,C 180,E1 4395.71,E2 4395.71} C_VEL
LIN {X 0,Y 522.881,Z 754.81,A -85,B 0,C 180,E1 4404.169,E2 4404.169} C_VEL
LIN {X 0,Y 522.515,Z 754.81,A -85,B 0,C 180,E1 4410.832,E2 4410.832} C_VEL
LIN {X 0,Y 522.745,Z 756.653,A -85,B 0,C 180,E1 4415.936,E2 4415.936} C_VEL
LIN {X 0,Y 525.456,Z 785.094,A -85,B 0,C 180,E1 4417.363,E2 4417.363} C_VEL
LIN {X 0,Y 524.277,Z 819.36,A -85,B 0,C 180,E1 4420.446,E2 4420.446} C_VEL
LIN {X 0,Y 523.624,Z 842.807,A -85,B 0,C 180,E1 4424.69,E2 4424.69} C_VEL
LIN {X 0,Y 523.289,Z 851.909,A -85,B 0,C 180,E1 4429.481,E2 4429.481} C_VEL
LIN {X 0,Y 523.704,Z 846.356,A -85,B 0,C 180,E1 4434.102,E2 4434.102} C_VEL
LIN {X 0,Y 524.132,Z 826.031,A -85,B 0,C 180,E1 4438.537,E2 4438.537} C_VEL
LIN {X 0,Y 525.203,Z 793.804,A -85,B 0,C 180,E1 4441.966,E2 4441.966} C_VEL
LIN {X 0,Y 523.809,Z 759.494,A -85,B 0,C 180,E1 4443.853,E2 4443.853} C_VEL
LIN {X 0,Y 522.75,Z 754.81,A -85,B 0,C 180,E1 4444.168,E2 4444.168} C_VEL
LIN {X 0,Y 522.261,Z 754.81,A -85,B 0,C 180,E1 4453.067,E2 4453.067} C_VEL
LIN {X 0,Y 522.089,Z 754.81,A -85,B 0,C 180,E1 4461.32,E2 4461.32} C_VEL
LIN {X 0,Y 522.339,Z 754.81,A -85,B 0,C 180,E1 4469.439,E2 4469.439} C_VEL
LIN {X 0,Y 522.222,Z 754.81,A -85,B 0,C 180,E1 4476.9,E2 4476.9} C_VEL
LIN {X 0,Y 522.574,Z 754.81,A -85,B 0,C 180,E1 4485.707,E2 4485.707} C_VEL
LIN {X 0,Y 522.858,Z 754.81,A -85,B 0,C 180,E1 4494.167,E2 4494.167} C_VEL
LIN {X 0,Y 523.011,Z 754.81,A -85,B 0,C 180,E1 4500.829,E2 4500.829} C_VEL
LIN {X 0,Y 522.724,Z 754.81,A -85,B 0,C 180,E1 4509.186,E2 4509.186} C_VEL
LIN {X 0,Y 522.6,Z 754.81,A -85,B 0,C 180,E1 4517.75,E2 4517.75} C_VEL
LIN {X 0,Y 522.623,Z 754.81,A -85,B 0,C 180,E1 4527.67,E2 4527.67} C_VEL
LIN {X 0,Y 522.464,Z 754.81,A -85,B 0,C 180,E1 4536.074,E2 4536.074} C_VEL
LIN {X 0,Y 514.333,Z 754.81,A -85,B 0,C 180,E1 4539.91,E2 4539.91} C_VEL
LIN {X 0,Y 514.281,Z 754.81,A -85,B 0,C 180,E1 4548.8,E2 4548.8} C_VEL
LIN {X 0,Y 514.22,Z 754.81,A -85,B 0,C 180,E1 4557.251,E2 4557.251} C_VEL
LIN {X 0,Y 514.762,Z 755.683,A -85,B 0,C 180,E1 4565.108,E2 4565.108} C_VEL
LIN {X 0,Y 522.168,Z 783.506,A -85,B 0,C 180,E1 4565.789,E2 4565.789} C_VEL
LIN {X 0,Y 521.557,Z 853.965,A -85,B 0,C 180,E1 4567.211,E2 4567.211} C_VEL
LIN {X 0,Y 519.584,Z 906.403,A -85,B 0,C 180,E1 4570.008,E2 4570.008} C_VEL
LIN {X 0,Y 517.518,Z 949.186,A -85,B 0,C 180,E1 4574.262,E2 4574.262} C_VEL
LIN {X 0,Y 516.057,Z 981.123,A -85,B 0,C 180,E1 4579.74,E2 4579.74} C_VEL
LIN {X 0,Y 515.259,Z 998.592,A -85,B 0,C 180,E1 4585.778,E2 4585.778} C_VEL
LIN {X 0,Y 515.302,Z 1001.836,A -85,B 0,C 180,E1 4590.844,E2 4590.844} C_VEL
LIN {X 0,Y 515.229,Z 994.252,A -85,B 0,C 180,E1 4596.342,E2 4596.342} C_VEL
LIN {X 0,Y 515.894,Z 973.563,A -85,B 0,C 180,E1 4601.884,E2 4601.884} C_VEL
LIN {X 0,Y 517.626,Z 938.836,A -85,B 0,C 180,E1 4606.998,E2 4606.998} C_VEL
LIN {X 0,Y 520.105,Z 895.061,A -85,B 0,C 180,E1 4610.771,E2 4610.771} C_VEL
LIN {X 0,Y 522.043,Z 842.58,A -85,B 0,C 180,E1 4613.162,E2 4613.162} C_VEL
LIN {X 0,Y 520.122,Z 771.402,A -85,B 0,C 180,E1 4614.469,E2 4614.469} C_VEL
LIN {X 0,Y 514.815,Z 754.81,A -85,B 0,C 180,E1 4615.013,E2 4615.013} C_VEL
LIN {X 0,Y 514.427,Z 754.81,A -85,B 0,C 180,E1 4625.118,E2 4625.118} C_VEL
LIN {X 0,Y 514.462,Z 754.81,A -85,B 0,C 180,E1 4633.886,E2 4633.886} C_VEL
LIN {X 0,Y 514.266,Z 754.81,A -85,B 0,C 180,E1 4644.245,E2 4644.245} C_VEL
LIN {X 0,Y 514.295,Z 754.81,A -85,B 0,C 180,E1 4654.158,E2 4654.158} C_VEL
LIN {X 0,Y 514.63,Z 754.81,A -85,B 0,C 180,E1 4663.734,E2 4663.734} C_VEL
LIN {X 0,Y 514.99,Z 754.81,A -85,B 0,C 180,E1 4672.382,E2 4672.382} C_VEL
LIN {X 0,Y 515.195,Z 754.81,A -85,B 0,C 180,E1 4682.535,E2 4682.535} C_VEL
LIN {X 0,Y 514.792,Z 754.81,A -85,B 0,C 180,E1 4691.049,E2 4691.049} C_VEL
LIN {X 0,Y 514.567,Z 754.81,A -85,B 0,C 180,E1 4699.828,E2 4699.828} C_VEL
LIN {X 0,Y 514.407,Z 754.81,A -85,B 0,C 180,E1 4709.506,E2 4709.506} C_VEL
LIN {X 0,Y 514.283,Z 754.81,A -85,B 0,C 180,E1 4719.38,E2 4719.38} C_VEL
LIN {X 0,Y 514.371,Z 754.81,A -85,B 0,C 180,E1 4728.795,E2 4728.795} C_VEL
LIN {X 0,Y 514.288,Z 754.81,A -85,B 0,C 180,E1 4738.909,E2 4738.909} C_VEL
LIN {X 0,Y 514.225,Z 754.81,A -85,B 0,C 180,E1 4746.521,E2 4746.521} C_VEL
LIN {X 0,Y 514.609,Z 754.81,A -85,B 0,C 180,E1 4755.483,E2 4755.483} C_VEL
LIN {X 0,Y 514.883,Z 754.81,A -85,B 0,C 180,E1 4764.078,E2 4764.078} C_VEL
LIN {X 0,Y 514.503,Z 754.81,A -85,B 0,C 180,E1 4770.844,E2 4770.844} C_VEL
LIN {X 0,Y 514.529,Z 756.279,A -85,B 0,C 180,E1 4775.606,E2 4775.606} C_VEL
LIN {X 0,Y 517.894,Z 784.731,A -85,B 0,C 180,E1 4777.048,E2 4777.048} C_VEL
LIN {X 0,Y 516.52,Z 819.657,A -85,B 0,C 180,E1 4780.174,E2 4780.174} C_VEL
LIN {X 0,Y 515.683,Z 843.189,A -85,B 0,C 180,E1 4784.485,E2 4784.485} C_VEL
LIN {X 0,Y 515.38,Z 851.392,A -85,B 0,C 180,E1 4788.009,E2 4788.009} C_VEL
LIN {X 0,Y 515.509,Z 850.371,A -85,B 0,C 180,E1 4792.629,E2 4792.629} C_VEL
LIN {X 0,Y 515.978,Z 836.123,A -85,B 0,C 180,E1 4797.121,E2 4797.121} C_VEL
LIN {X 0,Y 517.099,Z 808.25,A -85,B 0,C 180,E1 4801.032,E2 4801.032} C_VEL
LIN {X 0,Y 518.106,Z 770.295,A -85,B 0,C 180,E1 4803.65,E2 4803.65} C_VEL
LIN {X 0,Y 514.648,Z 754.81,A -85,B 0,C 180,E1 4804.622,E2 4804.622} C_VEL
LIN {X 0,Y 514.256,Z 754.81,A -85,B 0,C 180,E1 4813.906,E2 4813.906} C_VEL
LIN {X 0,Y 514.084,Z 754.81,A -85,B 0,C 180,E1 4822.758,E2 4822.758} C_VEL
LIN {X 0,Y 514.313,Z 754.81,A -85,B 0,C 180,E1 4830.864,E2 4830.864} C_VEL
LIN {X 0,Y 514.114,Z 754.81,A -85,B 0,C 180,E1 4840.154,E2 4840.154} C_VEL
LIN {X 0,Y 514.536,Z 754.81,A -85,B 0,C 180,E1 4848.945,E2 4848.945} C_VEL
LIN {X 0,Y 515.567,Z 754.81,A -85,B 0,C 180,E1 4859.155,E2 4859.155} C_VEL
LIN {X 0,Y 514.756,Z 754.81,A -85,B 0,C 180,E1 4869.026,E2 4869.026} C_VEL
LIN {X 0,Y 514.61,Z 754.81,A -85,B 0,C 180,E1 4878.035,E2 4878.035} C_VEL
LIN {X 0,Y 514.606,Z 754.81,A -85,B 0,C 180,E1 4887.197,E2 4887.197} C_VEL
LIN {X 0,Y 514.471,Z 754.81,A -85,B 0,C 180,E1 4897.204,E2 4897.204} C_VEL
LIN {X 0,Y 514.333,Z 754.81,A -85,B 0,C 180,E1 4899.91,E2 4899.91} C_VEL
LIN {X 0,Y 506.287,Z 754.81,A -85,B 0,C 180,E1 4903.809,E2 4903.809} C_VEL
LIN {X 0,Y 506.335,Z 754.81,A -85,B 0,C 180,E1 4914.237,E2 4914.237} C_VEL
LIN {X 0,Y 506.63,Z 754.81,A -85,B 0,C 180,E1 4924.535,E2 4924.535} C_VEL
LIN {X 0,Y 514.632,Z 786.352,A -85,B 0,C 180,E1 4925.542,E2 4925.542} C_VEL
LIN {X 0,Y 513.874,Z 854.232,A -85,B 0,C 180,E1 4926.965,E2 4926.965} C_VEL
LIN {X 0,Y 511.805,Z 905.662,A -85,B 0,C 180,E1 4929.76,E2 4929.76} C_VEL
LIN {X 0,Y 509.782,Z 947.489,A -85,B 0,C 180,E1 4933.795,E2 4933.795} C_VEL
LIN {X 0,Y 508.254,Z 979.181,A -85,B 0,C 180,E1 4939.132,E2 4939.132} C_VEL
LIN {X 0,Y 507.626,Z 997.046,A -85,B 0,C 180,E1 4944.855,E2 4944.855} C_VEL
LIN {X 0,Y 507.298,Z 1001.836,A -85,B 0,C 180,E1 4950.858,E2 4950.858} C_VEL
LIN {X 0,Y 507.238,Z 994.252,A -85,B 0,C 180,E1 4956.442,E2 4956.442} C_VEL
LIN {X 0,Y 507.958,Z 973.563,A -85,B 0,C 180,E1 4962.072,E2 4962.072} C_VEL
LIN {X 0,Y 509.814,Z 939.488,A -85,B 0,C 180,E1 4967.17,E2 4967.17} C_VEL
LIN {X 0,Y 512.418,Z 892.928,A -85,B 0,C 180,E1 4971.117,E2 4971.117} C_VEL
LIN {X 0,Y 514.508,Z 839.406,A -85,B 0,C 180,E1 4973.522,E2 4973.522} C_VEL
LIN {X 0,Y 512.449,Z 772.934,A -85,B 0,C 180,E1 4974.751,E2 4974.751} C_VEL
LIN {X 0,Y 506.765,Z 754.81,A -85,B 0,C 180,E1 4975.47,E2 4975.47} C_VEL
LIN {X 0,Y 506.447,Z 754.81,A -85,B 0,C 180,E1 4985.756,E2 4985.756} C_VEL
LIN {X 0,Y 506.316,Z 754.81,A -85,B 0,C 180,E1 4995.226,E2 4995.226} C_VEL
LIN {X 0,Y 506.289,Z 754.81,A -85,B 0,C 180,E1 5004.236,E2 5004.236} C_VEL
LIN {X 0,Y 506.296,Z 754.81,A -85,B 0,C 180,E1 5014.242,E2 5014.242} C_VEL
LIN {X 0,Y 506.609,Z 754.81,A -85,B 0,C 180,E1 5023.469,E2 5023.469} C_VEL
LIN {X 0,Y 506.958,Z 754.81,A -85,B 0,C 180,E1 5032.261,E2 5032.261} C_VEL
LIN {X 0,Y 507.194,Z 754.81,A -85,B 0,C 180,E1 5042.575,E2 5042.575} C_VEL
LIN {X 0,Y 506.765,Z 754.81,A -85,B 0,C 180,E1 5051.226,E2 5051.226} C_VEL
LIN {X 0,Y 506.578,Z 754.81,A -85,B 0,C 180,E1 5060.154,E2 5060.154} C_VEL
LIN {X 0,Y 506.418,Z 754.81,A -85,B 0,C 180,E1 5069.636,E2 5069.636} C_VEL
LIN {X 0,Y 506.237,Z 754.81,A -85,B 0,C 180,E1 5080.143,E2 5080.143} C_VEL
LIN {X 0,Y 506.187,Z 754.81,A -85,B 0,C 180,E1 5089.865,E2 5089.865} C_VEL
LIN {X 0,Y 506.277,Z 754.81,A -85,B 0,C 180,E1 5098.684,E2 5098.684} C_VEL
LIN {X 0,Y 505.998,Z 754.81,A -85,B 0,C 180,E1 5107.981,E2 5107.981} C_VEL
LIN {X 0,Y 506.447,Z 754.81,A -85,B 0,C 180,E1 5117.012,E2 5117.012} C_VEL
LIN {X 0,Y 506.837,Z 754.81,A -85,B 0,C 180,E1 5125.707,E2 5125.707} C_VEL
LIN {X 0,Y 506.064,Z 754.81,A -85,B 0,C 180,E1 5132.578,E2 5132.578} C_VEL
LIN {X 0,Y 506.555,Z 756.806,A -85,B 0,C 180,E1 5135.305,E2 5135.305} C_VEL
LIN {X 0,Y 510.293,Z 784.392,A -85,B 0,C 180,E1 5136.724,E2 5136.724} C_VEL
LIN {X 0,Y 508.75,Z 819.98,A -85,B 0,C 180,E1 5139.898,E2 5139.898} C_VEL
LIN {X 0,Y 507.822,Z 843.552,A -85,B 0,C 180,E1 5144.161,E2 5144.161} C_VEL
LIN {X 0,Y 507.451,Z 852.889,A -85,B 0,C 180,E1 5148.301,E2 5148.301} C_VEL
LIN {X 0,Y 507.663,Z 851.223,A -85,B 0,C 180,E1 5152.868,E2 5152.868} C_VEL
LIN {X 0,Y 508.376,Z 835.762,A -85,B 0,C 180,E1 5157.561,E2 5157.561} C_VEL
LIN {X 0,Y 509.508,Z 807.557,A -85,B 0,C 180,E1 5161.415,E2 5161.415} C_VEL
LIN {X 0,Y 510.083,Z 769.274,A -85,B 0,C 180,E1 5164.026,E2 5164.026} C_VEL
LIN {X 0,Y 506.611,Z 754.81,A -85,B 0,C 180,E1 5164.851,E2 5164.851} C_VEL
LIN {X 0,Y 506.222,Z 754.81,A -85,B 0,C 180,E1 5174.788,E2 5174.788} C_VEL
LIN {X 0,Y 506.203,Z 754.81,A -85,B 0,C 180,E1 5184.223,E2 5184.223} C_VEL
LIN {X 0,Y 506.513,Z 754.81,A -85,B 0,C 180,E1 5194.249,E2 5194.249} C_VEL
LIN {X 0,Y 506.592,Z 754.81,A -85,B 0,C 180,E1 5205.246,E2 5205.246} C_VEL
LIN {X 0,Y 506.86,Z 754.81,A -85,B 0,C 180,E1 5213.983,E2 5213.983} C_VEL
LIN {X 0,Y 507.005,Z 754.81,A -85,B 0,C 180,E1 5220.855,E2 5220.855} C_VEL
LIN {X 0,Y 506.721,Z 754.81,A -85,B 0,C 180,E1 5229.479,E2 5229.479} C_VEL
LIN {X 0,Y 506.683,Z 754.81,A -85,B 0,C 180,E1 5239.36,E2 5239.36} C_VEL
LIN {X 0,Y 506.475,Z 754.81,A -85,B 0,C 180,E1 5249.627,E2 5249.627} C_VEL
LIN {X 0,Y 506.449,Z 754.81,A -85,B 0,C 180,E1 5257.896,E2 5257.896} C_VEL
LIN {X 0,Y 506.287,Z 754.81,A -85,B 0,C 180,E1 5263.809,E2 5263.809} C_VEL
LIN {X 0,Y 498.159,Z 754.81,A -85,B 0,C 180,E1 5267.763,E2 5267.763} C_VEL
LIN {X 0,Y 498.158,Z 754.81,A -85,B 0,C 180,E1 5276.898,E2 5276.898} C_VEL
LIN {X 0,Y 498.762,Z 756.155,A -85,B 0,C 180,E1 5284.463,E2 5284.463} C_VEL
LIN {X 0,Y 507.095,Z 788.129,A -85,B 0,C 180,E1 5285.272,E2 5285.272} C_VEL
LIN {X 0,Y 506.216,Z 854.475,A -85,B 0,C 180,E1 5286.713,E2 5286.713} C_VEL
LIN {X 0,Y 503.954,Z 906.083,A -85,B 0,C 180,E1 5289.603,E2 5289.603} C_VEL
LIN {X 0,Y 501.736,Z 949.804,A -85,B 0,C 180,E1 5293.979,E2 5293.979} C_VEL
LIN {X 0,Y 500.316,Z 979.688,A -85,B 0,C 180,E1 5299.072,E2 5299.072} C_VEL
LIN {X 0,Y 499.653,Z 997.045,A -85,B 0,C 180,E1 5304.773,E2 5304.773} C_VEL
LIN {X 0,Y 499.295,Z 1001.836,A -85,B 0,C 180,E1 5310.871,E2 5310.871} C_VEL
LIN {X 0,Y 499.227,Z 994.252,A -85,B 0,C 180,E1 5316.546,E2 5316.546} C_VEL
LIN {X 0,Y 500.025,Z 973.533,A -85,B 0,C 180,E1 5322.267,E2 5322.267} C_VEL
LIN {X 0,Y 501.871,Z 939.703,A -85,B 0,C 180,E1 5327.264,E2 5327.264} C_VEL
LIN {X 0,Y 504.619,Z 893.511,A -85,B 0,C 180,E1 5331.301,E2 5331.301} C_VEL
LIN {X 0,Y 506.891,Z 840.192,A -85,B 0,C 180,E1 5333.781,E2 5333.781} C_VEL
LIN {X 0,Y 505.071,Z 775.04,A -85,B 0,C 180,E1 5335.022,E2 5335.022} C_VEL
LIN {X 0,Y 498.755,Z 754.81,A -85,B 0,C 180,E1 5335.652,E2 5335.652} C_VEL
LIN {X 0,Y 498.43,Z 754.81,A -85,B 0,C 180,E1 5346.422,E2 5346.422} C_VEL
LIN {X 0,Y 498.2,Z 754.81,A -85,B 0,C 180,E1 5356.739,E2 5356.739} C_VEL
LIN {X 0,Y 498.144,Z 754.81,A -85,B 0,C 180,E1 5365.699,E2 5365.699} C_VEL
LIN {X 0,Y 498.294,Z 754.81,A -85,B 0,C 180,E1 5373.954,E2 5373.954} C_VEL
LIN {X 0,Y 498.614,Z 754.81,A -85,B 0,C 180,E1 5383.484,E2 5383.484} C_VEL
LIN {X 0,Y 499.212,Z 754.81,A -85,B 0,C 180,E1 5393.895,E2 5393.895} C_VEL
LIN {X 0,Y 499.174,Z 754.81,A -85,B 0,C 180,E1 5402.616,E2 5402.616} C_VEL
LIN {X 0,Y 498.741,Z 754.81,A -85,B 0,C 180,E1 5411.409,E2 5411.409} C_VEL
LIN {X 0,Y 498.559,Z 754.81,A -85,B 0,C 180,E1 5420.492,E2 5420.492} C_VEL
LIN {X 0,Y 498.366,Z 754.81,A -85,B 0,C 180,E1 5430.164,E2 5430.164} C_VEL
LIN {X 0,Y 498.135,Z 754.81,A -85,B 0,C 180,E1 5440.922,E2 5440.922} C_VEL
LIN {X 0,Y 498.139,Z 754.81,A -85,B 0,C 180,E1 5449.08,E2 5449.08} C_VEL
LIN {X 0,Y 498.229,Z 754.81,A -85,B 0,C 180,E1 5457.788,E2 5457.788} C_VEL
LIN {X 0,Y 498.275,Z 754.81,A -85,B 0,C 180,E1 5465.721,E2 5465.721} C_VEL
LIN {X 0,Y 498.603,Z 754.81,A -85,B 0,C 180,E1 5475.006,E2 5475.006} C_VEL
LIN {X 0,Y 498.884,Z 754.81,A -85,B 0,C 180,E1 5483.888,E2 5483.888} C_VEL
LIN {X 0,Y 498.501,Z 754.81,A -85,B 0,C 180,E1 5490.872,E2 5490.872} C_VEL
LIN {X 0,Y 498.426,Z 756.623,A -85,B 0,C 180,E1 5494.967,E2 5494.967} C_VEL
LIN {X 0,Y 502.706,Z 783.954,A -85,B 0,C 180,E1 5496.391,E2 5496.391} C_VEL
LIN {X 0,Y 501.026,Z 820.107,A -85,B 0,C 180,E1 5499.589,E2 5499.589} C_VEL
LIN {X 0,Y 499.978,Z 844.537,A -85,B 0,C 180,E1 5504.009,E2 5504.009} C_VEL
LIN {X 0,Y 499.548,Z 854.367,A -85,B 0,C 180,E1 5508.601,E2 5508.601} C_VEL
LIN {X 0,Y 499.918,Z 850.875,A -85,B 0,C 180,E1 5513.717,E2 5513.717} C_VEL
LIN {X 0,Y 500.766,Z 833.189,A -85,B 0,C 180,E1 5518.408,E2 5518.408} C_VEL
LIN {X 0,Y 502.131,Z 803.142,A -85,B 0,C 180,E1 5522.147,E2 5522.147} C_VEL
LIN {X 0,Y 501.234,Z 765.026,A -85,B 0,C 180,E1 5524.578,E2 5524.578} C_VEL
LIN {X 0,Y 498.548,Z 754.81,A -85,B 0,C 180,E1 5525.189,E2 5525.189} C_VEL
LIN {X 0,Y 498.214,Z 754.81,A -85,B 0,C 180,E1 5535.709,E2 5535.709} C_VEL
LIN {X 0,Y 498.298,Z 754.81,A -85,B 0,C 180,E1 5545.705,E2 5545.705} C_VEL
LIN {X 0,Y 498.32,Z 754.81,A -85,B 0,C 180,E1 5555.722,E2 5555.722} C_VEL
LIN {X 0,Y 498.573,Z 754.81,A -85,B 0,C 180,E1 5565.004,E2 5565.004} C_VEL
LIN {X 0,Y 498.859,Z 754.81,A -85,B 0,C 180,E1 5573.886,E2 5573.886} C_VEL
LIN {X 0,Y 498.999,Z 754.81,A -85,B 0,C 180,E1 5580.869,E2 5580.869} C_VEL
LIN {X 0,Y 498.726,Z 754.81,A -85,B 0,C 180,E1 5589.632,E2 5589.632} C_VEL
LIN {X 0,Y 498.631,Z 754.81,A -85,B 0,C 180,E1 5598.634,E2 5598.634} C_VEL
LIN {X 0,Y 498.493,Z 754.81,A -85,B 0,C 180,E1 5608.153,E2 5608.153} C_VEL
LIN {X 0,Y 498.327,Z 754.81,A -85,B 0,C 180,E1 5618.627,E2 5618.627} C_VEL
LIN {X 0,Y 498.159,Z 754.81,A -85,B 0,C 180,E1 5627.763,E2 5627.763} C_VEL
LIN {X 0,Y 490.196,Z 754.81,A -85,B 0,C 180,E1 5631.784,E2 5631.784} C_VEL
LIN {X 0,Y 490.565,Z 754.81,A -85,B 0,C 180,E1 5641.836,E2 5641.836} C_VEL
LIN {X 0,Y 490.77,Z 756.416,A -85,B 0,C 180,E1 5644.124,E2 5644.124} C_VEL
LIN {X 0,Y 499.576,Z 788.429,A -85,B 0,C 180,E1 5644.973,E2 5644.973} C_VEL
LIN {X 0,Y 498.64,Z 853.261,A -85,B 0,C 180,E1 5646.397,E2 5646.397} C_VEL
LIN {X 0,Y 496.188,Z 904.925,A -85,B 0,C 180,E1 5649.319,E2 5649.319} C_VEL
LIN {X 0,Y 493.826,Z 948.353,A -85,B 0,C 180,E1 5653.715,E2 5653.715} C_VEL
LIN {X 0,Y 492.234,Z 980.893,A -85,B 0,C 180,E1 5659.34,E2 5659.34} C_VEL
LIN {X 0,Y 491.669,Z 997.044,A -85,B 0,C 180,E1 5664.688,E2 5664.688} C_VEL
LIN {X 0,Y 491.312,Z 1001.836,A -85,B 0,C 180,E1 5670.885,E2 5670.885} C_VEL
LIN {X 0,Y 491.228,Z 994.187,A -85,B 0,C 180,E1 5676.653,E2 5676.653} C_VEL
LIN {X 0,Y 492.024,Z 973.549,A -85,B 0,C 180,E1 5682.243,E2 5682.243} C_VEL
LIN {X 0,Y 493.99,Z 938.831,A -85,B 0,C 180,E1 5687.482,E2 5687.482} C_VEL
LIN {X 0,Y 496.894,Z 892.059,A -85,B 0,C 180,E1 5691.622,E2 5691.622} C_VEL
LIN {X 0,Y 499.295,Z 838.967,A -85,B 0,C 180,E1 5694.107,E2 5694.107} C_VEL
LIN {X 0,Y 497.744,Z 777.47,A -85,B 0,C 180,E1 5695.293,E2 5695.293} C_VEL
LIN {X 0,Y 490.726,Z 754.81,A -85,B 0,C 180,E1 5696.056,E2 5696.056} C_VEL
LIN {X 0,Y 490.318,Z 754.81,A -85,B 0,C 180,E1 5704.932,E2 5704.932} C_VEL
LIN {X 0,Y 490.27,Z 754.81,A -85,B 0,C 180,E1 5714.145,E2 5714.145} C_VEL
LIN {X 0,Y 490.194,Z 754.81,A -85,B 0,C 180,E1 5722.869,E2 5722.869} C_VEL
LIN {X 0,Y 490.249,Z 754.81,A -85,B 0,C 180,E1 5733.333,E2 5733.333} C_VEL
LIN {X 0,Y 490.571,Z 754.81,A -85,B 0,C 180,E1 5742.912,E2 5742.912} C_VEL
LIN {X 0,Y 490.916,Z 754.81,A -85,B 0,C 180,E1 5752.006,E2 5752.006} C_VEL
LIN {X 0,Y 491.175,Z 754.81,A -85,B 0,C 180,E1 5762.659,E2 5762.659} C_VEL
LIN {X 0,Y 490.721,Z 754.81,A -85,B 0,C 180,E1 5771.598,E2 5771.598} C_VEL
LIN {X 0,Y 490.566,Z 754.81,A -85,B 0,C 180,E1 5780.842,E2 5780.842} C_VEL
LIN {X 0,Y 490.262,Z 754.81,A -85,B 0,C 180,E1 5790.716,E2 5790.716} C_VEL
LIN {X 0,Y 490.116,Z 754.81,A -85,B 0,C 180,E1 5800.657,E2 5800.657} C_VEL
LIN {X 0,Y 490.012,Z 754.81,A -85,B 0,C 180,E1 5810.588,E2 5810.588} C_VEL
LIN {X 0,Y 490.171,Z 754.81,A -85,B 0,C 180,E1 5819.279,E2 5819.279} C_VEL
LIN {X 0,Y 489.994,Z 754.81,A -85,B 0,C 180,E1 5829.134,E2 5829.134} C_VEL
LIN {X 0,Y 490.485,Z 754.81,A -85,B 0,C 180,E1 5838.397,E2 5838.397} C_VEL
LIN {X 0,Y 491.182,Z 754.81,A -85,B 0,C 180,E1 5847.343,E2 5847.343} C_VEL
LIN {X 0,Y 490.402,Z 756.816,A -85,B 0,C 180,E1 5854.631,E2 5854.631} C_VEL
LIN {X 0,Y 495.093,Z 785.368,A -85,B 0,C 180,E1 5856.158,E2 5856.158} C_VEL
LIN {X 0,Y 493.334,Z 820.399,A -85,B 0,C 180,E1 5859.293,E2 5859.293} C_VEL
LIN {X 0,Y 492.143,Z 845.128,A -85,B 0,C 180,E1 5863.746,E2 5863.746} C_VEL
LIN {X 0,Y 491.623,Z 855.741,A -85,B 0,C 180,E1 5868.912,E2 5868.912} C_VEL
LIN {X 0,Y 492.093,Z 850.348,A -85,B 0,C 180,E1 5874.525,E2 5874.525} C_VEL
LIN {X 0,Y 493.056,Z 830.175,A -85,B 0,C 180,E1 5879.282,E2 5879.282} C_VEL
LIN {X 0,Y 494.682,Z 797.81,A -85,B 0,C 180,E1 5882.933,E2 5882.933} C_VEL
LIN {X 0,Y 493.571,Z 766.407,A -85,B 0,C 180,E1 5884.857,E2 5884.857} C_VEL
LIN {X 0,Y 490.524,Z 754.81,A -85,B 0,C 180,E1 5885.454,E2 5885.454} C_VEL
LIN {X 0,Y 490.213,Z 754.81,A -85,B 0,C 180,E1 5895.848,E2 5895.848} C_VEL
LIN {X 0,Y 490.205,Z 754.81,A -85,B 0,C 180,E1 5905.122,E2 5905.122} C_VEL
LIN {X 0,Y 490.338,Z 754.81,A -85,B 0,C 180,E1 5915.301,E2 5915.301} C_VEL
LIN {X 0,Y 490.584,Z 754.81,A -85,B 0,C 180,E1 5924.753,E2 5924.753} C_VEL
LIN {X 0,Y 490.873,Z 754.81,A -85,B 0,C 180,E1 5933.786,E2 5933.786} C_VEL
LIN {X 0,Y 491.015,Z 754.81,A -85,B 0,C 180,E1 5940.883,E2 5940.883} C_VEL
LIN {X 0,Y 490.714,Z 754.81,A -85,B 0,C 180,E1 5949.791,E2 5949.791} C_VEL
LIN {X 0,Y 490.585,Z 754.81,A -85,B 0,C 180,E1 5959.356,E2 5959.356} C_VEL
LIN {X 0,Y 490.448,Z 754.81,A -85,B 0,C 180,E1 5968.657,E2 5968.657} C_VEL
LIN {X 0,Y 490.289,Z 754.81,A -85,B 0,C 180,E1 5977.881,E2 5977.881} C_VEL
LIN {X 0,Y 490.162,Z 754.81,A -85,B 0,C 180,E1 5987.765,E2 5987.765} C_VEL
LIN {X 0,Y 490.196,Z 754.81,A -85,B 0,C 180,E1 5991.784,E2 5991.784} C_VEL
LIN {X 0,Y 482.071,Z 754.81,A -85,B 0,C 180,E1 5995.874,E2 5995.874} C_VEL
LIN {X 0,Y 482.632,Z 755.916,A -85,B 0,C 180,E1 6003.748,E2 6003.748} C_VEL
LIN {X 0,Y 492.075,Z 789.431,A -85,B 0,C 180,E1 6004.674,E2 6004.674} C_VEL
LIN {X 0,Y 491.01,Z 853.421,A -85,B 0,C 180,E1 6006.125,E2 6006.125} C_VEL
LIN {X 0,Y 488.336,Z 905.707,A -85,B 0,C 180,E1 6009.18,E2 6009.18} C_VEL
LIN {X 0,Y 485.851,Z 948.586,A -85,B 0,C 180,E1 6013.674,E2 6013.674} C_VEL
LIN {X 0,Y 484.309,Z 979.607,A -85,B 0,C 180,E1 6019.164,E2 6019.164} C_VEL
LIN {X 0,Y 483.412,Z 997.728,A -85,B 0,C 180,E1 6025.499,E2 6025.499} C_VEL
LIN {X 0,Y 483.333,Z 1001.188,A -85,B 0,C 180,E1 6030.9,E2 6030.9} C_VEL
LIN {X 0,Y 483.268,Z 993.081,A -85,B 0,C 180,E1 6036.763,E2 6036.763} C_VEL
LIN {X 0,Y 484.078,Z 972.262,A -85,B 0,C 180,E1 6042.447,E2 6042.447} C_VEL
LIN {X 0,Y 486.114,Z 938.049,A -85,B 0,C 180,E1 6047.695,E2 6047.695} C_VEL
LIN {X 0,Y 489.18,Z 891.303,A -85,B 0,C 180,E1 6051.907,E2 6051.907} C_VEL
LIN {X 0,Y 491.723,Z 838.665,A -85,B 0,C 180,E1 6054.414,E2 6054.414} C_VEL
LIN {X 0,Y 489.969,Z 778.607,A -85,B 0,C 180,E1 6055.612,E2 6055.612} C_VEL
LIN {X 0,Y 482.694,Z 754.81,A -85,B 0,C 180,E1 6056.366,E2 6056.366} C_VEL
LIN {X 0,Y 482.28,Z 754.81,A -85,B 0,C 180,E1 6066.645,E2 6066.645} C_VEL
LIN {X 0,Y 482.196,Z 754.81,A -85,B 0,C 180,E1 6075.083,E2 6075.083} C_VEL
LIN {X 0,Y 482.099,Z 754.81,A -85,B 0,C 180,E1 6084.387,E2 6084.387} C_VEL
LIN {X 0,Y 482.204,Z 754.81,A -85,B 0,C 180,E1 6093.76,E2 6093.76} C_VEL
LIN {X 0,Y 482.591,Z 754.81,A -85,B 0,C 180,E1 6103.562,E2 6103.562} C_VEL
LIN {X 0,Y 483.149,Z 754.81,A -85,B 0,C 180,E1 6113.691,E2 6113.691} C_VEL
LIN {X 0,Y 483.155,Z 754.81,A -85,B 0,C 180,E1 6122.703,E2 6122.703} C_VEL
LIN {X 0,Y 482.738,Z 754.81,A -85,B 0,C 180,E1 6131.793,E2 6131.793} C_VEL
LIN {X 0,Y 482.531,Z 754.81,A -85,B 0,C 180,E1 6141.205,E2 6141.205} C_VEL
LIN {X 0,Y 482.222,Z 754.81,A -85,B 0,C 180,E1 6151.285,E2 6151.285} C_VEL
LIN {X 0,Y 482.103,Z 754.81,A -85,B 0,C 180,E1 6160.191,E2 6160.191} C_VEL
LIN {X 0,Y 482.011,Z 754.81,A -85,B 0,C 180,E1 6170.479,E2 6170.479} C_VEL
LIN {X 0,Y 482.167,Z 754.81,A -85,B 0,C 180,E1 6180.8,E2 6180.8} C_VEL
LIN {X 0,Y 482.166,Z 754.81,A -85,B 0,C 180,E1 6190.702,E2 6190.702} C_VEL
LIN {X 0,Y 482.823,Z 754.81,A -85,B 0,C 180,E1 6200.045,E2 6200.045} C_VEL
LIN {X 0,Y 483.371,Z 754.81,A -85,B 0,C 180,E1 6209.1,E2 6209.1} C_VEL
LIN {X 0,Y 482.117,Z 755.599,A -85,B 0,C 180,E1 6214.23,E2 6214.23} C_VEL
LIN {X 0,Y 487.493,Z 786.778,A -85,B 0,C 180,E1 6215.918,E2 6215.918} C_VEL
LIN {X 0,Y 485.546,Z 822.448,A -85,B 0,C 180,E1 6219.217,E2 6219.217} C_VEL
LIN {X 0,Y 484.305,Z 846.13,A -85,B 0,C 180,E1 6223.592,E2 6223.592} C_VEL
LIN {X 0,Y 483.886,Z 855.372,A -85,B 0,C 180,E1 6227.333,E2 6227.333} C_VEL
LIN {X 0,Y 483.99,Z 854.725,A -85,B 0,C 180,E1 6233.075,E2 6233.075} C_VEL
LIN {X 0,Y 484.95,Z 839.337,A -85,B 0,C 180,E1 6237.995,E2 6237.995} C_VEL
LIN {X 0,Y 486.495,Z 811.321,A -85,B 0,C 180,E1 6242.049,E2 6242.049} C_VEL
LIN {X 0,Y 487.131,Z 772.567,A -85,B 0,C 180,E1 6244.877,E2 6244.877} C_VEL
LIN {X 0,Y 482.487,Z 754.81,A -85,B 0,C 180,E1 6245.871,E2 6245.871} C_VEL
LIN {X 0,Y 482.136,Z 754.81,A -85,B 0,C 180,E1 6255.089,E2 6255.089} C_VEL
LIN {X 0,Y 482.059,Z 754.81,A -85,B 0,C 180,E1 6264.378,E2 6264.378} C_VEL
LIN {X 0,Y 482.345,Z 754.81,A -85,B 0,C 180,E1 6273.724,E2 6273.724} C_VEL
LIN {X 0,Y 482.543,Z 754.81,A -85,B 0,C 180,E1 6284.493,E2 6284.493} C_VEL
LIN {X 0,Y 482.869,Z 754.81,A -85,B 0,C 180,E1 6293.683,E2 6293.683} C_VEL
LIN {X 0,Y 483.009,Z 754.81,A -85,B 0,C 180,E1 6300.898,E2 6300.898} C_VEL
LIN {X 0,Y 482.719,Z 754.81,A -85,B 0,C 180,E1 6309.955,E2 6309.955} C_VEL
LIN {X 0,Y 482.599,Z 754.81,A -85,B 0,C 180,E1 6319.277,E2 6319.277} C_VEL
LIN {X 0,Y 482.349,Z 754.81,A -85,B 0,C 180,E1 6329.184,E2 6329.184} C_VEL
LIN {X 0,Y 482.277,Z 754.81,A -85,B 0,C 180,E1 6339.563,E2 6339.563} C_VEL
LIN {X 0,Y 482.19,Z 754.81,A -85,B 0,C 180,E1 6349.821,E2 6349.821} C_VEL
LIN {X 0,Y 482.071,Z 754.81,A -85,B 0,C 180,E1 6355.874,E2 6355.874} C_VEL
LIN {X 0,Y 474.27,Z 754.81,A -85,B 0,C 180,E1 6360.028,E2 6360.028} C_VEL
LIN {X 0,Y 474.717,Z 756.545,A -85,B 0,C 180,E1 6363.386,E2 6363.386} C_VEL
LIN {X 0,Y 484.597,Z 791.719,A -85,B 0,C 180,E1 6364.382,E2 6364.382} C_VEL
LIN {X 0,Y 483.379,Z 853.575,A -85,B 0,C 180,E1 6365.844,E2 6365.844} C_VEL
LIN {X 0,Y 480.534,Z 905.383,A -85,B 0,C 180,E1 6368.947,E2 6368.947} C_VEL
LIN {X 0,Y 477.884,Z 948.815,A -85,B 0,C 180,E1 6373.631,E2 6373.631} C_VEL
LIN {X 0,Y 476.22,Z 980.15,A -85,B 0,C 180,E1 6379.442,E2 6379.442} C_VEL
LIN {X 0,Y 475.527,Z 996.532,A -85,B 0,C 180,E1 6385.424,E2 6385.424} C_VEL
LIN {X 0,Y 475.43,Z 1000.013,A -85,B 0,C 180,E1 6390.915,E2 6390.915} C_VEL
LIN {X 0,Y 475.323,Z 991.875,A -85,B 0,C 180,E1 6396.877,E2 6396.877} C_VEL
LIN {X 0,Y 476.151,Z 971.018,A -85,B 0,C 180,E1 6402.649,E2 6402.649} C_VEL
LIN {X 0,Y 478.278,Z 936.614,A -85,B 0,C 180,E1 6407.991,E2 6407.991} C_VEL
LIN {X 0,Y 481.43,Z 891.556,A -85,B 0,C 180,E1 6412.133,E2 6412.133} C_VEL
LIN {X 0,Y 484.188,Z 838.648,A -85,B 0,C 180,E1 6414.722,E2 6414.722} C_VEL
LIN {X 0,Y 482.464,Z 780.26,A -85,B 0,C 180,E1 6415.92,E2 6415.92} C_VEL
LIN {X 0,Y 474.641,Z 754.81,A -85,B 0,C 180,E1 6416.827,E2 6416.827} C_VEL
LIN {X 0,Y 474.25,Z 754.81,A -85,B 0,C 180,E1 6426.299,E2 6426.299} C_VEL
LIN {X 0,Y 474.071,Z 754.81,A -85,B 0,C 180,E1 6436.513,E2 6436.513} C_VEL
LIN {X 0,Y 474.057,Z 754.81,A -85,B 0,C 180,E1 6445.933,E2 6445.933} C_VEL
LIN {X 0,Y 474.176,Z 754.81,A -85,B 0,C 180,E1 6455.802,E2 6455.802} C_VEL
LIN {X 0,Y 474.638,Z 754.81,A -85,B 0,C 180,E1 6464.233,E2 6464.233} C_VEL
LIN {X 0,Y 475.118,Z 754.81,A -85,B 0,C 180,E1 6473.584,E2 6473.584} C_VEL
LIN {X 0,Y 475.134,Z 754.81,A -85,B 0,C 180,E1 6482.748,E2 6482.748} C_VEL
LIN {X 0,Y 474.701,Z 754.81,A -85,B 0,C 180,E1 6492.822,E2 6492.822} C_VEL
LIN {X 0,Y 474.522,Z 754.81,A -85,B 0,C 180,E1 6501.581,E2 6501.581} C_VEL
LIN {X 0,Y 474.118,Z 754.81,A -85,B 0,C 180,E1 6511.98,E2 6511.98} C_VEL
LIN {X 0,Y 474.018,Z 754.81,A -85,B 0,C 180,E1 6521.204,E2 6521.204} C_VEL
LIN {X 0,Y 473.965,Z 754.81,A -85,B 0,C 180,E1 6531.364,E2 6531.364} C_VEL
LIN {X 0,Y 474.145,Z 754.81,A -85,B 0,C 180,E1 6541.667,E2 6541.667} C_VEL
LIN {X 0,Y 474.383,Z 754.81,A -85,B 0,C 180,E1 6552.307,E2 6552.307} C_VEL
LIN {X 0,Y 475.022,Z 754.81,A -85,B 0,C 180,E1 6561.734,E2 6561.734} C_VEL
LIN {X 0,Y 474.465,Z 754.81,A -85,B 0,C 180,E1 6570.916,E2 6570.916} C_VEL
LIN {X 0,Y 474.225,Z 756.37,A -85,B 0,C 180,E1 6573.899,E2 6573.899} C_VEL
LIN {X 0,Y 479.975,Z 786.299,A -85,B 0,C 180,E1 6575.556,E2 6575.556} C_VEL
LIN {X 0,Y 477.901,Z 822.101,A -85,B 0,C 180,E1 6578.82,E2 6578.82} C_VEL
LIN {X 0,Y 476.511,Z 846.484,A -85,B 0,C 180,E1 6583.259,E2 6583.259} C_VEL
LIN {X 0,Y 475.938,Z 857.001,A -85,B 0,C 180,E1 6587.632,E2 6587.632} C_VEL
LIN {X 0,Y 476.041,Z 856.592,A -85,B 0,C 180,E1 6592.686,E2 6592.686} C_VEL
LIN {X 0,Y 476.996,Z 841.821,A -85,B 0,C 180,E1 6597.872,E2 6597.872} C_VEL
LIN {X 0,Y 478.694,Z 814.391,A -85,B 0,C 180,E1 6602.085,E2 6602.085} C_VEL
LIN {X 0,Y 479.879,Z 775.531,A -85,B 0,C 180,E1 6605.074,E2 6605.074} C_VEL
LIN {X 0,Y 474.444,Z 754.81,A -85,B 0,C 180,E1 6606.28,E2 6606.28} C_VEL
LIN {X 0,Y 474.086,Z 754.81,A -85,B 0,C 180,E1 6616.508,E2 6616.508} C_VEL
LIN {X 0,Y 474.108,Z 754.81,A -85,B 0,C 180,E1 6625.931,E2 6625.931} C_VEL
LIN {X 0,Y 474.137,Z 754.81,A -85,B 0,C 180,E1 6635.81,E2 6635.81} C_VEL
LIN {X 0,Y 474.443,Z 754.81,A -85,B 0,C 180,E1 6646.117,E2 6646.117} C_VEL
LIN {X 0,Y 474.821,Z 754.81,A -85,B 0,C 180,E1 6655.415,E2 6655.415} C_VEL
LIN {X 0,Y 474.803,Z 754.81,A -85,B 0,C 180,E1 6662.746,E2 6662.746} C_VEL
LIN {X 0,Y 474.758,Z 754.81,A -85,B 0,C 180,E1 6672.857,E2 6672.857} C_VEL
LIN {X 0,Y 474.517,Z 754.81,A -85,B 0,C 180,E1 6681.576,E2 6681.576} C_VEL
LIN {X 0,Y 474.185,Z 754.81,A -85,B 0,C 180,E1 6691.995,E2 6691.995} C_VEL
LIN {X 0,Y 474.175,Z 754.81,A -85,B 0,C 180,E1 6701.228,E2 6701.228} C_VEL
LIN {X 0,Y 474.206,Z 754.81,A -85,B 0,C 180,E1 6711.629,E2 6711.629} C_VEL
LIN {X 0,Y 474.27,Z 754.81,A -85,B 0,C 180,E1 6720.028,E2 6720.028} C_VEL
LIN {X 0,Y 466.476,Z 754.81,A -85,B 0,C 180,E1 6722.793,E2 6722.793} C_VEL
LIN {X 0,Y 477.176,Z 795.625,A -85,B 0,C 180,E1 6724.105,E2 6724.105} C_VEL
LIN {X 0,Y 475.694,Z 855.664,A -85,B 0,C 180,E1 6725.629,E2 6725.629} C_VEL
LIN {X 0,Y 472.616,Z 906.739,A -85,B 0,C 180,E1 6728.844,E2 6728.844} C_VEL
LIN {X 0,Y 469.897,Z 949.042,A -85,B 0,C 180,E1 6733.586,E2 6733.586} C_VEL
LIN {X 0,Y 468.3,Z 978.863,A -85,B 0,C 180,E1 6739.262,E2 6739.262} C_VEL
LIN {X 0,Y 467.623,Z 995.332,A -85,B 0,C 180,E1 6745.347,E2 6745.347} C_VEL
LIN {X 0,Y 467.511,Z 998.834,A -85,B 0,C 180,E1 6750.931,E2 6750.931} C_VEL
LIN {X 0,Y 467.378,Z 990.79,A -85,B 0,C 180,E1 6756.944,E2 6756.944} C_VEL
LIN {X 0,Y 468.266,Z 969.054,A -85,B 0,C 180,E1 6763.006,E2 6763.006} C_VEL
LIN {X 0,Y 470.488,Z 933.879,A -85,B 0,C 180,E1 6768.452,E2 6768.452} C_VEL
LIN {X 0,Y 473.871,Z 888.337,A -85,B 0,C 180,E1 6772.601,E2 6772.601} C_VEL
LIN {X 0,Y 476.777,Z 834.996,A -85,B 0,C 180,E1 6775.141,E2 6775.141} C_VEL
LIN {X 0,Y 475.041,Z 782.206,A -85,B 0,C 180,E1 6776.224,E2 6776.224} C_VEL
LIN {X 0,Y 466.601,Z 754.81,A -85,B 0,C 180,E1 6777.138,E2 6777.138} C_VEL
LIN {X 0,Y 466.174,Z 754.81,A -85,B 0,C 180,E1 6787.107,E2 6787.107} C_VEL
LIN {X 0,Y 466.005,Z 754.81,A -85,B 0,C 180,E1 6797.116,E2 6797.116} C_VEL
LIN {X 0,Y 466.047,Z 754.81,A -85,B 0,C 180,E1 6807.505,E2 6807.505} C_VEL
LIN {X 0,Y 466.348,Z 754.81,A -85,B 0,C 180,E1 6818.04,E2 6818.04} C_VEL
LIN {X 0,Y 466.827,Z 754.81,A -85,B 0,C 180,E1 6827.804,E2 6827.804} C_VEL
LIN {X 0,Y 466.815,Z 754.81,A -85,B 0,C 180,E1 6837.207,E2 6837.207} C_VEL
LIN {X 0,Y 466.815,Z 754.81,A -85,B 0,C 180,E1 6844.664,E2 6844.664} C_VEL
LIN {X 0,Y 466.74,Z 754.81,A -85,B 0,C 180,E1 6854.116,E2 6854.116} C_VEL
LIN {X 0,Y 466.431,Z 754.81,A -85,B 0,C 180,E1 6864,E2 6864} C_VEL
LIN {X 0,Y 465.97,Z 754.81,A -85,B 0,C 180,E1 6873.85,E2 6873.85} C_VEL
LIN {X 0,Y 465.951,Z 754.81,A -85,B 0,C 180,E1 6884.449,E2 6884.449} C_VEL
LIN {X 0,Y 466.04,Z 754.81,A -85,B 0,C 180,E1 6895.259,E2 6895.259} C_VEL
LIN {X 0,Y 466.169,Z 754.81,A -85,B 0,C 180,E1 6903.929,E2 6903.929} C_VEL
LIN {X 0,Y 466.486,Z 754.81,A -85,B 0,C 180,E1 6913.947,E2 6913.947} C_VEL
LIN {X 0,Y 466.89,Z 754.81,A -85,B 0,C 180,E1 6923.467,E2 6923.467} C_VEL
LIN {X 0,Y 466.453,Z 754.81,A -85,B 0,C 180,E1 6930.931,E2 6930.931} C_VEL
LIN {X 0,Y 466.124,Z 755.713,A -85,B 0,C 180,E1 6933.499,E2 6933.499} C_VEL
LIN {X 0,Y 472.353,Z 788.354,A -85,B 0,C 180,E1 6935.343,E2 6935.343} C_VEL
LIN {X 0,Y 470.113,Z 824.082,A -85,B 0,C 180,E1 6938.729,E2 6938.729} C_VEL
LIN {X 0,Y 468.622,Z 848.39,A -85,B 0,C 180,E1 6943.341,E2 6943.341} C_VEL
LIN {X 0,Y 467.992,Z 858.549,A -85,B 0,C 180,E1 6947.942,E2 6947.942} C_VEL
LIN {X 0,Y 468.328,Z 855.895,A -85,B 0,C 180,E1 6953.894,E2 6953.894} C_VEL
LIN {X 0,Y 469.522,Z 839.867,A -85,B 0,C 180,E1 6958.699,E2 6958.699} C_VEL
LIN {X 0,Y 471.38,Z 811.561,A -85,B 0,C 180,E1 6962.753,E2 6962.753} C_VEL
LIN {X 0,Y 471.283,Z 772.776,A -85,B 0,C 180,E1 6965.636,E2 6965.636} C_VEL
LIN {X 0,Y 466.352,Z 754.81,A -85,B 0,C 180,E1 6966.756,E2 6966.756} C_VEL
LIN {X 0,Y 466.017,Z 754.81,A -85,B 0,C 180,E1 6977.113,E2 6977.113} C_VEL
LIN {X 0,Y 466.103,Z 754.81,A -85,B 0,C 180,E1 6987.503,E2 6987.503} C_VEL
LIN {X 0,Y 466.13,Z 754.81,A -85,B 0,C 180,E1 6995.984,E2 6995.984} C_VEL
LIN {X 0,Y 466.425,Z 754.81,A -85,B 0,C 180,E1 7005.874,E2 7005.874} C_VEL
LIN {X 0,Y 466.814,Z 754.81,A -85,B 0,C 180,E1 7015.336,E2 7015.336} C_VEL
LIN {X 0,Y 466.803,Z 754.81,A -85,B 0,C 180,E1 7022.793,E2 7022.793} C_VEL
LIN {X 0,Y 466.79,Z 754.81,A -85,B 0,C 180,E1 7032.197,E2 7032.197} C_VEL
LIN {X 0,Y 466.451,Z 754.81,A -85,B 0,C 180,E1 7041.994,E2 7041.994} C_VEL
LIN {X 0,Y 466.143,Z 754.81,A -85,B 0,C 180,E1 7052.488,E2 7052.488} C_VEL
LIN {X 0,Y 466.103,Z 754.81,A -85,B 0,C 180,E1 7062.898,E2 7062.898} C_VEL
LIN {X 0,Y 466.105,Z 754.81,A -85,B 0,C 180,E1 7072.963,E2 7072.963} C_VEL
LIN {X 0,Y 466.476,Z 754.81,A -85,B 0,C 180,E1 7082.793,E2 7082.793} C_VEL
LIN {X 0,Y 471.095,Z 765.935,A -85,B 0,C 180,E1 7083.359,E2 7083.359} C_VEL
LIN {X 0,Y 469.386,Z 789.52,A -85,B 0,C 180,E1 7083.645,E2 7083.645} C_VEL
LIN {X 0,Y 468.411,Z 851.043,A -85,B 0,C 180,E1 7085.132,E2 7085.132} C_VEL
LIN {X 0,Y 465.139,Z 902.73,A -85,B 0,C 180,E1 7088.288,E2 7088.288} C_VEL
LIN {X 0,Y 462.036,Z 946.257,A -85,B 0,C 180,E1 7093.107,E2 7093.107} C_VEL
LIN {X 0,Y 460.391,Z 977.577,A -85,B 0,C 180,E1 7099.075,E2 7099.075} C_VEL
LIN {X 0,Y 459.708,Z 994.129,A -85,B 0,C 180,E1 7105.267,E2 7105.267} C_VEL
LIN {X 0,Y 459.606,Z 997.658,A -85,B 0,C 180,E1 7110.947,E2 7110.947} C_VEL
LIN {X 0,Y 459.458,Z 989.021,A -85,B 0,C 180,E1 7117.288,E2 7117.288} C_VEL
LIN {X 0,Y 460.437,Z 967.073,A -85,B 0,C 180,E1 7123.38,E2 7123.38} C_VEL
LIN {X 0,Y 462.825,Z 931.426,A -85,B 0,C 180,E1 7128.893,E2 7128.893} C_VEL
LIN {X 0,Y 466.384,Z 884.619,A -85,B 0,C 180,E1 7133.111,E2 7133.111} C_VEL
LIN {X 0,Y 469.39,Z 832.062,A -85,B 0,C 180,E1 7135.546,E2 7135.546} C_VEL
LIN {X 0,Y 467.477,Z 783.535,A -85,B 0,C 180,E1 7136.556,E2 7136.556} C_VEL
LIN {X 0,Y 458.537,Z 754.81,A -85,B 0,C 180,E1 7137.699,E2 7137.699} C_VEL
LIN {X 0,Y 458.08,Z 754.81,A -85,B 0,C 180,E1 7148.879,E2 7148.879} C_VEL
LIN {X 0,Y 457.984,Z 754.81,A -85,B 0,C 180,E1 7158.208,E2 7158.208} C_VEL
LIN {X 0,Y 458.085,Z 754.81,A -85,B 0,C 180,E1 7169.107,E2 7169.107} C_VEL
LIN {X 0,Y 458.431,Z 754.81,A -85,B 0,C 180,E1 7179.663,E2 7179.663} C_VEL
LIN {X 0,Y 458.709,Z 754.81,A -85,B 0,C 180,E1 7189.519,E2 7189.519} C_VEL
LIN {X 0,Y 459.017,Z 754.81,A -85,B 0,C 180,E1 7199.055,E2 7199.055} C_VEL
LIN {X 0,Y 459.027,Z 754.81,A -85,B 0,C 180,E1 7208.558,E2 7208.558} C_VEL
LIN {X 0,Y 458.558,Z 754.81,A -85,B 0,C 180,E1 7218.327,E2 7218.327} C_VEL
LIN {X 0,Y 458.175,Z 754.81,A -85,B 0,C 180,E1 7228.705,E2 7228.705} C_VEL
LIN {X 0,Y 457.887,Z 754.81,A -85,B 0,C 180,E1 7238.843,E2 7238.843} C_VEL
LIN {X 0,Y 457.945,Z 754.81,A -85,B 0,C 180,E1 7248.215,E2 7248.215} C_VEL
LIN {X 0,Y 458.043,Z 754.81,A -85,B 0,C 180,E1 7259.099,E2 7259.099} C_VEL
LIN {X 0,Y 457.936,Z 754.81,A -85,B 0,C 180,E1 7267.597,E2 7267.597} C_VEL
LIN {X 0,Y 458.435,Z 754.81,A -85,B 0,C 180,E1 7277.574,E2 7277.574} C_VEL
LIN {X 0,Y 459.129,Z 754.81,A -85,B 0,C 180,E1 7287.158,E2 7287.158} C_VEL
LIN {X 0,Y 458.244,Z 756.41,A -85,B 0,C 180,E1 7293.141,E2 7293.141} C_VEL
LIN {X 0,Y 464.729,Z 790.353,A -85,B 0,C 180,E1 7295.126,E2 7295.126} C_VEL
LIN {X 0,Y 462.353,Z 826.153,A -85,B 0,C 180,E1 7298.648,E2 7298.648} C_VEL
LIN {X 0,Y 460.73,Z 850.313,A -85,B 0,C 180,E1 7303.45,E2 7303.45} C_VEL
LIN {X 0,Y 460.056,Z 860.049,A -85,B 0,C 180,E1 7308.262,E2 7308.262} C_VEL
LIN {X 0,Y 460.515,Z 856.411,A -85,B 0,C 180,E1 7314.325,E2 7314.325} C_VEL
LIN {X 0,Y 461.904,Z 838.123,A -85,B 0,C 180,E1 7319.462,E2 7319.462} C_VEL
LIN {X 0,Y 464.115,Z 807.791,A -85,B 0,C 180,E1 7323.506,E2 7323.506} C_VEL
LIN {X 0,Y 463.455,Z 773.179,A -85,B 0,C 180,E1 7326.018,E2 7326.018} C_VEL
LIN {X 0,Y 458.277,Z 754.81,A -85,B 0,C 180,E1 7327.281,E2 7327.281} C_VEL
LIN {X 0,Y 457.986,Z 754.81,A -85,B 0,C 180,E1 7338.206,E2 7338.206} C_VEL
LIN {X 0,Y 458.108,Z 754.81,A -85,B 0,C 180,E1 7349.103,E2 7349.103} C_VEL
LIN {X 0,Y 457.973,Z 754.81,A -85,B 0,C 180,E1 7357.598,E2 7357.598} C_VEL
LIN {X 0,Y 458.392,Z 754.81,A -85,B 0,C 180,E1 7367.589,E2 7367.589} C_VEL
LIN {X 0,Y 459.223,Z 754.81,A -85,B 0,C 180,E1 7377.865,E2 7377.865} C_VEL
LIN {X 0,Y 458.803,Z 754.81,A -85,B 0,C 180,E1 7388.557,E2 7388.557} C_VEL
LIN {X 0,Y 458.466,Z 754.81,A -85,B 0,C 180,E1 7398.325,E2 7398.325} C_VEL
LIN {X 0,Y 458.254,Z 754.81,A -85,B 0,C 180,E1 7408.694,E2 7408.694} C_VEL
LIN {X 0,Y 458.096,Z 754.81,A -85,B 0,C 180,E1 7418.877,E2 7418.877} C_VEL
LIN {X 0,Y 458.015,Z 754.81,A -85,B 0,C 180,E1 7428.198,E2 7428.198} C_VEL
LIN {X 0,Y 458.141,Z 754.81,A -85,B 0,C 180,E1 7439.108,E2 7439.108} C_VEL
LIN {X 0,Y 458.59,Z 756.284,A -85,B 0,C 180,E1 7442.566,E2 7442.566} C_VEL
LIN {X 0,Y 469.386,Z 789.52,A -85,B 0,C 180,E1 7443.645,E2 7443.645} C_VEL
LIN {X 0,Y 467.308,Z 806.572,A -85,B 0,C 180,E1 7443.812,E2 7443.812} C_VEL
LIN {X 0,Y 462.051,Z 824.283,A -85,B 0,C 180,E1 7443.921,E2 7443.921} C_VEL
LIN {X 0,Y 459.273,Z 876.439,A -85,B 0,C 180,E1 7446.124,E2 7446.124} C_VEL
LIN {X 0,Y 455.467,Z 924.197,A -85,B 0,C 180,E1 7450.158,E2 7450.158} C_VEL
LIN {X 0,Y 452.739,Z 961.914,A -85,B 0,C 180,E1 7455.67,E2 7455.67} C_VEL
LIN {X 0,Y 451.763,Z 984.322,A -85,B 0,C 180,E1 7461.306,E2 7461.306} C_VEL
LIN {X 0,Y 451.564,Z 995.236,A -85,B 0,C 180,E1 7467.111,E2 7467.111} C_VEL
LIN {X 0,Y 451.876,Z 994.313,A -85,B 0,C 180,E1 7473.852,E2 7473.852} C_VEL
LIN {X 0,Y 452.158,Z 978.276,A -85,B 0,C 180,E1 7480.638,E2 7480.638} C_VEL
LIN {X 0,Y 453.872,Z 947.682,A -85,B 0,C 180,E1 7486.83,E2 7486.83} C_VEL
LIN {X 0,Y 457.269,Z 904.827,A -85,B 0,C 180,E1 7491.809,E2 7491.809} C_VEL
LIN {X 0,Y 460.699,Z 854.492,A -85,B 0,C 180,E1 7495.067,E2 7495.067} C_VEL
LIN {X 0,Y 462.271,Z 795.163,A -85,B 0,C 180,E1 7496.622,E2 7496.622} C_VEL
LIN {X 0,Y 450.511,Z 754.81,A -85,B 0,C 180,E1 7497.966,E2 7497.966} C_VEL
LIN {X 0,Y 450.07,Z 754.81,A -85,B 0,C 180,E1 7508.595,E2 7508.595} C_VEL
LIN {X 0,Y 449.983,Z 754.81,A -85,B 0,C 180,E1 7519.361,E2 7519.361} C_VEL
LIN {X 0,Y 450.078,Z 754.81,A -85,B 0,C 180,E1 7529.296,E2 7529.296} C_VEL
LIN {X 0,Y 450.356,Z 754.81,A -85,B 0,C 180,E1 7539.282,E2 7539.282} C_VEL
LIN {X 0,Y 450.719,Z 754.81,A -85,B 0,C 180,E1 7549.331,E2 7549.331} C_VEL
LIN {X 0,Y 451.011,Z 754.81,A -85,B 0,C 180,E1 7559.038,E2 7559.038} C_VEL
LIN {X 0,Y 451.002,Z 754.81,A -85,B 0,C 180,E1 7568.712,E2 7568.712} C_VEL
LIN {X 0,Y 450.549,Z 754.81,A -85,B 0,C 180,E1 7578.664,E2 7578.664} C_VEL
LIN {X 0,Y 450.091,Z 754.81,A -85,B 0,C 180,E1 7589.27,E2 7589.27} C_VEL
LIN {X 0,Y 449.927,Z 754.81,A -85,B 0,C 180,E1 7600.631,E2 7600.631} C_VEL
LIN {X 0,Y 449.918,Z 754.81,A -85,B 0,C 180,E1 7609.372,E2 7609.372} C_VEL
LIN {X 0,Y 450.018,Z 754.81,A -85,B 0,C 180,E1 7619.311,E2 7619.311} C_VEL
LIN {X 0,Y 449.93,Z 754.81,A -85,B 0,C 180,E1 7629.258,E2 7629.258} C_VEL
LIN {X 0,Y 450.638,Z 754.81,A -85,B 0,C 180,E1 7639.325,E2 7639.325} C_VEL
LIN {X 0,Y 451.339,Z 754.81,A -85,B 0,C 180,E1 7649.036,E2 7649.036} C_VEL
LIN {X 0,Y 450.117,Z 755.341,A -85,B 0,C 180,E1 7652.717,E2 7652.717} C_VEL
LIN {X 0,Y 457.242,Z 790.309,A -85,B 0,C 180,E1 7654.759,E2 7654.759} C_VEL
LIN {X 0,Y 454.769,Z 825.27,A -85,B 0,C 180,E1 7658.153,E2 7658.153} C_VEL
LIN {X 0,Y 452.977,Z 850.016,A -85,B 0,C 180,E1 7662.901,E2 7662.901} C_VEL
LIN {X 0,Y 452.348,Z 859.891,A -85,B 0,C 180,E1 7667.027,E2 7667.027} C_VEL
LIN {X 0,Y 452.363,Z 860.365,A -85,B 0,C 180,E1 7672.693,E2 7672.693} C_VEL
LIN {X 0,Y 453.496,Z 846.374,A -85,B 0,C 180,E1 7678.148,E2 7678.148} C_VEL
LIN {X 0,Y 455.632,Z 819.624,A -85,B 0,C 180,E1 7682.646,E2 7682.646} C_VEL
LIN {X 0,Y 457.704,Z 782.217,A -85,B 0,C 180,E1 7685.84,E2 7685.84} C_VEL
LIN {X 0,Y 450.215,Z 754.81,A -85,B 0,C 180,E1 7687.612,E2 7687.612} C_VEL
LIN {X 0,Y 449.982,Z 754.81,A -85,B 0,C 180,E1 7696.476,E2 7696.476} C_VEL
LIN {X 0,Y 449.958,Z 754.81,A -85,B 0,C 180,E1 7706.184,E2 7706.184} C_VEL
LIN {X 0,Y 450.082,Z 754.81,A -85,B 0,C 180,E1 7715.07,E2 7715.07} C_VEL
LIN {X 0,Y 450.374,Z 754.81,A -85,B 0,C 180,E1 7725.359,E2 7725.359} C_VEL
LIN {X 0,Y 450.799,Z 754.81,A -85,B 0,C 180,E1 7735.17,E2 7735.17} C_VEL
LIN {X 0,Y 450.821,Z 754.81,A -85,B 0,C 180,E1 7742.892,E2 7742.892} C_VEL
LIN {X 0,Y 450.77,Z 754.81,A -85,B 0,C 180,E1 7752.638,E2 7752.638} C_VEL
LIN {X 0,Y 450.37,Z 754.81,A -85,B 0,C 180,E1 7762.796,E2 7762.796} C_VEL
LIN {X 0,Y 450.047,Z 754.81,A -85,B 0,C 180,E1 7773.803,E2 7773.803} C_VEL
LIN {X 0,Y 450.041,Z 754.81,A -85,B 0,C 180,E1 7783.727,E2 7783.727} C_VEL
LIN {X 0,Y 449.996,Z 754.81,A -85,B 0,C 180,E1 7793.831,E2 7793.831} C_VEL
LIN {X 0,Y 450.475,Z 755.655,A -85,B 0,C 180,E1 7802.112,E2 7802.112} C_VEL
LIN {X 0,Y 462.311,Z 796.409,A -85,B 0,C 180,E1 7803.408,E2 7803.408} C_VEL
LIN {X 0,Y 462.051,Z 824.283,A -85,B 0,C 180,E1 7803.921,E2 7803.921} C_VEL
LIN {X 0,Y 452.795,Z 857.855,A -85,B 0,C 180,E1 7804.779,E2 7804.779} C_VEL
LIN {X 0,Y 449.085,Z 908.297,A -85,B 0,C 180,E1 7808.316,E2 7808.316} C_VEL
LIN {X 0,Y 445.961,Z 949.503,A -85,B 0,C 180,E1 7813.442,E2 7813.442} C_VEL
LIN {X 0,Y 444.259,Z 978.509,A -85,B 0,C 180,E1 7819.669,E2 7819.669} C_VEL
LIN {X 0,Y 443.756,Z 993.029,A -85,B 0,C 180,E1 7826.079,E2 7826.079} C_VEL
LIN {X 0,Y 443.777,Z 995.305,A -85,B 0,C 180,E1 7830.98,E2 7830.98} C_VEL
LIN {X 0,Y 443.592,Z 988.118,A -85,B 0,C 180,E1 7836.878,E2 7836.878} C_VEL
LIN {X 0,Y 444.455,Z 966.941,A -85,B 0,C 180,E1 7843.33,E2 7843.33} C_VEL
LIN {X 0,Y 446.946,Z 932.403,A -85,B 0,C 180,E1 7849.076,E2 7849.076} C_VEL
LIN {X 0,Y 450.864,Z 885.98,A -85,B 0,C 180,E1 7853.56,E2 7853.56} C_VEL
LIN {X 0,Y 454.29,Z 833.214,A -85,B 0,C 180,E1 7856.191,E2 7856.191} C_VEL
